C05458=1071.279,380.940,394.327,175.389,32.950,156.009
C05459=1071.272,380.693,394.366,175.385,32.942,156.008
C05460=1071.265,380.447,394.406,175.380,32.935,156.006
C05461=1071.258,380.200,394.445,175.376,32.928,156.005
C05462=1071.252,379.953,394.483,175.372,32.922,156.003
C05463=1071.245,379.706,394.522,175.368,32.915,156.002
C05464=1071.238,379.459,394.561,175.363,32.908,156.001
C05465=1071.231,379.213,394.600,175.359,32.901,155.999
C05466=1071.224,378.966,394.639,175.355,32.894,155.998
C05467=1071.217,378.719,394.678,175.350,32.887,155.996
C05468=1071.211,378.472,394.717,175.346,32.880,155.995
C05469=1071.204,378.225,394.755,175.342,32.874,155.993
C05470=1071.197,377.979,394.794,175.338,32.867,155.992
C05471=1071.190,377.732,394.833,175.333,32.860,155.990
C05472=1071.183,377.485,394.872,175.329,32.853,155.989
C05473=1071.178,377.238,394.910,175.325,32.846,155.988
C05474=1071.170,376.992,394.948,175.321,32.839,155.986
C05475=1071.163,376.745,394.987,175.316,32.832,155.985
C05476=1071.156,376.498,395.026,175.312,32.826,155.983
C05477=1071.150,376.251,395.064,175.308,32.819,155.982
C05478=1071.143,376.004,395.102,175.304,32.812,155.980
C05479=1071.136,375.757,395.141,175.300,32.806,155.979
C05480=1071.129,375.510,395.180,175.295,32.799,155.978
C05481=1071.123,375.263,395.218,175.291,32.792,155.976
C05482=1071.117,375.017,395.257,175.287,32.785,155.975
C05483=1071.110,374.770,395.296,175.283,32.779,155.973
C05484=1071.103,374.522,395.334,175.279,32.772,155.972
C05485=1071.097,374.276,395.372,175.274,32.766,155.971
C05486=1071.090,374.029,395.410,175.270,32.759,155.969
C05487=1071.083,373.782,395.449,175.266,32.753,155.968
C05488=1071.077,373.535,395.487,175.262,32.746,155.966
C05489=1071.070,373.288,395.526,175.258,32.740,155.965
C05490=1071.062,372.987,395.572,175.253,32.731,155.963
C05491=1071.054,372.685,395.619,175.248,32.723,155.962
C05492=1071.045,372.384,395.665,175.243,32.715,155.960
C05493=1071.037,372.082,395.711,175.237,32.708,155.959
C05494=1071.028,371.755,395.762,175.232,32.699,155.957
C05495=1071.019,371.427,395.812,175.227,32.691,155.955
C05496=1071.012,371.180,395.850,175.222,32.684,155.954
C05497=1071.006,370.934,395.888,175.218,32.678,155.952
C05498=1070.999,370.686,395.927,175.215,32.671,155.951
C05499=1070.992,370.439,395.964,175.211,32.665,155.950
C05500=1070.986,370.192,396.002,175.207,32.659,155.948
C05501=1070.979,369.945,396.039,175.203,32.652,155.947
C05502=1070.972,369.698,396.078,175.199,32.646,155.946
C05503=1070.966,369.452,396.115,175.195,32.640,155.944
C05504=1070.959,369.204,396.153,175.190,32.633,155.943
C05505=1070.953,368.957,396.192,175.186,32.627,155.942
C05506=1070.946,368.711,396.229,175.182,32.621,155.940
C05507=1070.939,368.463,396.267,175.178,32.614,155.939
C05508=1070.933,368.217,396.304,175.174,32.608,155.938
C05509=1070.926,367.969,396.342,175.170,32.602,155.937
C05510=1070.919,367.722,396.380,175.166,32.596,155.935
C05511=1070.913,367.475,396.417,175.162,32.589,155.934
C05512=1070.906,367.228,396.455,175.158,32.583,155.933
C05513=1070.900,366.982,396.493,175.154,32.577,155.931
C05514=1070.893,366.734,396.530,175.150,32.571,155.930
C05515=1070.887,366.487,396.567,175.146,32.564,155.929
C05516=1070.880,366.240,396.605,175.143,32.558,155.928
C05517=1070.874,365.993,396.643,175.139,32.552,155.926
C05518=1070.867,365.746,396.680,175.135,32.546,155.925
C05519=1070.861,365.499,396.718,175.131,32.539,155.924
C05520=1070.854,365.251,396.755,175.126,32.534,155.923
C05521=1070.848,365.005,396.792,175.122,32.527,155.921
C05522=1070.841,364.758,396.830,175.118,32.521,155.920
C05523=1070.835,364.510,396.867,175.114,32.515,155.919
C05524=1070.828,364.263,396.905,175.110,32.509,155.918
C05525=1070.821,364.017,396.942,175.106,32.503,155.916
C05526=1070.814,363.769,396.978,175.102,32.497,155.915
C05527=1070.808,363.522,397.016,175.098,32.490,155.914
C05528=1070.801,363.274,397.053,175.094,32.485,155.913
C05529=1070.795,363.028,397.090,175.091,32.479,155.911
C05530=1070.789,362.780,397.128,175.087,32.472,155.910
C05531=1070.782,362.533,397.165,175.083,32.467,155.909
C05532=1070.776,362.286,397.201,175.079,32.461,155.908
C05533=1070.768,362.039,397.239,175.075,32.455,155.907
C05534=1070.762,361.792,397.275,175.071,32.449,155.905
C05535=1070.756,361.545,397.313,175.067,32.443,155.904
C05536=1070.749,361.298,397.350,175.063,32.437,155.903
C05537=1070.742,361.050,397.387,175.060,32.431,155.902
C05538=1070.736,360.804,397.424,175.056,32.425,155.900
C05539=1070.729,360.557,397.460,175.052,32.419,155.899
C05540=1070.723,360.308,397.498,175.049,32.413,155.898
C05541=1070.716,360.062,397.535,175.045,32.408,155.897
C05542=1070.710,359.815,397.571,175.041,32.402,155.896
C05543=1070.703,359.567,397.608,175.037,32.396,155.895
C05544=1070.697,359.343,397.641,175.033,32.391,155.893
C05545=1070.692,359.119,397.675,175.030,32.385,155.892
C05546=1070.686,358.895,397.708,175.026,32.379,155.891
C05547=1070.680,358.671,397.741,175.023,32.374,155.890
C05548=1070.674,358.447,397.774,175.019,32.369,155.889
C05549=1070.668,358.223,397.807,175.015,32.364,155.888
C05550=1070.661,357.998,397.841,175.013,32.359,155.887
C05551=1070.656,357.774,397.875,175.009,32.354,155.886
C05552=1070.650,357.527,397.911,175.005,32.348,155.885
C05553=1070.644,357.280,397.947,175.001,32.342,155.884
C05554=1070.637,357.032,397.984,174.998,32.336,155.882
C05555=1070.630,356.786,398.020,174.994,32.331,155.881
C05556=1070.623,356.539,398.057,174.990,32.325,155.880
C05557=1070.617,356.291,398.093,174.986,32.319,155.879
C05558=1070.610,356.044,398.130,174.982,32.314,155.878
C05559=1070.604,355.797,398.166,174.979,32.308,155.877
C05560=1070.597,355.550,398.203,174.975,32.302,155.876
C05561=1070.591,355.303,398.239,174.971,32.296,155.874
C05562=1070.584,355.055,398.276,174.967,32.291,155.873
C05563=1070.578,354.807,398.312,174.964,32.285,155.872
C05564=1070.572,354.560,398.348,174.960,32.279,155.871
C05565=1070.565,354.313,398.385,174.956,32.274,155.870
C05566=1070.559,354.066,398.421,174.952,32.268,155.869
C05567=1070.553,353.819,398.457,174.949,32.262,155.868
C05568=1070.547,353.571,398.493,174.945,32.256,155.867
C05569=1070.540,353.323,398.530,174.941,32.251,155.866
C05570=1070.533,353.077,398.566,174.938,32.245,155.864
C05571=1070.527,352.829,398.602,174.934,32.240,155.863
C05572=1070.520,352.582,398.638,174.930,32.234,155.862
C05573=1070.514,352.335,398.674,174.926,32.229,155.861
C05574=1070.508,352.087,398.710,174.923,32.223,155.860
C05575=1070.502,351.840,398.747,174.919,32.217,155.859
C05576=1070.494,351.593,398.782,174.916,32.212,155.858
C05577=1070.488,351.346,398.818,174.912,32.207,155.857
C05578=1070.482,351.098,398.855,174.908,32.201,155.856
C05579=1070.475,350.851,398.890,174.904,32.195,155.854
C05580=1070.468,350.604,398.927,174.900,32.190,155.853
C05581=1070.462,350.356,398.962,174.897,32.184,155.852
C05582=1070.455,350.109,398.998,174.894,32.179,155.851
C05583=1070.449,349.862,399.034,174.890,32.174,155.850
C05584=1070.443,349.614,399.070,174.886,32.168,155.849
C05585=1070.437,349.367,399.106,174.882,32.163,155.848
C05586=1070.430,349.119,399.141,174.878,32.157,155.847
C05587=1070.424,348.872,399.177,174.875,32.152,155.846
C05588=1070.417,348.625,399.213,174.872,32.146,155.845
C05589=1070.411,348.377,399.249,174.868,32.141,155.844
C05590=1070.405,348.130,399.284,174.864,32.136,155.843
C05591=1070.398,347.883,399.320,174.861,32.130,155.842
C05592=1070.392,347.635,399.356,174.857,32.125,155.840
C05593=1070.386,347.388,399.392,174.853,32.119,155.839
C05594=1070.379,347.140,399.427,174.849,32.114,155.838
C05595=1070.373,346.893,399.463,174.847,32.109,155.837
C05596=1070.366,346.646,399.498,174.843,32.103,155.836
C05597=1070.360,346.398,399.534,174.839,32.098,155.835
C05598=1070.354,346.151,399.569,174.835,32.093,155.834
C05599=1070.348,345.904,399.604,174.832,32.087,155.833
C05600=1070.342,345.681,399.637,174.828,32.083,155.832
C05601=1070.336,345.459,399.668,174.825,32.078,155.831
C05602=1070.331,345.237,399.700,174.823,32.073,155.830
C05603=1070.325,345.014,399.732,174.819,32.068,155.829
C05604=1070.319,344.792,399.764,174.816,32.064,155.828
C05605=1070.314,344.570,399.796,174.812,32.059,155.828
C05606=1070.307,344.347,399.827,174.809,32.054,155.827
C05607=1070.302,344.125,399.859,174.806,32.049,155.826
C05608=1070.296,343.877,399.895,174.803,32.044,155.825
C05609=1070.289,343.630,399.930,174.799,32.038,155.824
C05610=1070.283,343.383,399.965,174.796,32.033,155.823
C05611=1070.277,343.136,400.000,174.792,32.028,155.822
C05612=1070.270,342.888,400.035,174.788,32.023,155.821
C05613=1070.263,342.641,400.071,174.785,32.018,155.819
C05614=1070.257,342.393,400.106,174.782,32.013,155.819
C05615=1070.251,342.145,400.141,174.778,32.007,155.818
C05616=1070.244,341.898,400.176,174.774,32.002,155.816
C05617=1070.238,341.651,400.211,174.771,31.997,155.816
C05618=1070.232,341.403,400.246,174.767,31.992,155.814
C05619=1070.225,341.155,400.281,174.763,31.986,155.813
C05620=1070.219,340.908,400.317,174.761,31.982,155.812
C05621=1070.212,340.660,400.352,174.757,31.976,155.811
C05622=1070.206,340.414,400.386,174.753,31.971,155.811
C05623=1070.200,340.166,400.421,174.750,31.966,155.809
C05624=1070.194,339.918,400.457,174.746,31.961,155.808
C05625=1070.188,339.671,400.491,174.742,31.956,155.808
C05626=1070.181,339.423,400.526,174.740,31.950,155.806
C05627=1070.175,339.176,400.561,174.736,31.946,155.806
C05628=1070.169,338.928,400.596,174.732,31.940,155.804
C05629=1070.162,338.681,400.631,174.729,31.935,155.804
C05630=1070.156,338.433,400.665,174.725,31.930,155.803
C05631=1070.150,338.185,400.701,174.722,31.925,155.802
C05632=1070.144,337.938,400.735,174.719,31.920,155.801
C05633=1070.137,337.691,400.770,174.715,31.915,155.800
C05634=1070.131,337.443,400.804,174.712,31.910,155.799
C05635=1070.125,337.196,400.839,174.708,31.905,155.798
C05636=1070.118,336.948,400.874,174.704,31.900,155.797
C05637=1070.112,336.701,400.909,174.702,31.895,155.796
C05638=1070.106,336.454,400.943,174.698,31.890,155.795
C05639=1070.099,336.206,400.977,174.695,31.885,155.794
C05640=1070.092,335.958,401.012,174.691,31.880,155.793
C05641=1070.087,335.711,401.046,174.687,31.875,155.792
C05642=1070.080,335.463,401.081,174.685,31.870,155.791
C05643=1070.074,335.215,401.117,174.681,31.865,155.790
C05644=1070.068,334.968,401.151,174.678,31.860,155.789
C05645=1070.062,334.720,401.185,174.674,31.855,155.788
C05646=1070.056,334.473,401.219,174.670,31.850,155.787
C05647=1070.049,334.225,401.254,174.667,31.845,155.786
C05648=1070.043,333.977,401.289,174.664,31.840,155.785
C05649=1070.037,333.730,401.323,174.661,31.835,155.784
C05650=1070.030,333.482,401.357,174.657,31.830,155.783
C05651=1070.024,333.235,401.391,174.654,31.825,155.782
C05652=1070.017,332.987,401.425,174.650,31.820,155.781
C05653=1070.011,332.740,401.460,174.647,31.815,155.781
C05654=1070.005,332.492,401.494,174.644,31.810,155.779
C05655=1069.999,332.245,401.528,174.640,31.805,155.779
C05656=1069.993,332.020,401.560,174.637,31.801,155.778
C05657=1069.987,331.795,401.591,174.634,31.797,155.777
C05658=1069.981,331.570,401.622,174.632,31.792,155.776
C05659=1069.977,331.345,401.653,174.628,31.788,155.775
C05660=1069.971,331.121,401.684,174.625,31.783,155.774
C05661=1069.965,330.896,401.715,174.622,31.779,155.773
C05662=1069.959,330.671,401.746,174.619,31.774,155.773
C05663=1069.953,330.446,401.777,174.617,31.770,155.772
C05664=1069.947,330.199,401.811,174.613,31.765,155.771
C05665=1069.940,329.951,401.844,174.609,31.760,155.770
C05666=1069.934,329.703,401.878,174.606,31.755,155.769
C05667=1069.928,329.455,401.912,174.602,31.751,155.768
C05668=1069.921,329.208,401.946,174.600,31.746,155.767
C05669=1069.915,328.960,401.980,174.596,31.741,155.766
C05670=1069.908,328.713,402.014,174.593,31.737,155.766
C05671=1069.902,328.465,402.047,174.589,31.732,155.765
C05672=1069.896,328.217,402.081,174.586,31.727,155.764
C05673=1069.889,327.970,402.115,174.583,31.722,155.763
C05674=1069.883,327.723,402.149,174.580,31.718,155.762
C05675=1069.876,327.474,402.182,174.576,31.713,155.761
C05676=1069.870,327.227,402.217,174.573,31.708,155.760
C05677=1069.864,326.979,402.251,174.569,31.704,155.759
C05678=1069.858,326.731,402.284,174.567,31.699,155.758
C05679=1069.852,326.484,402.318,174.563,31.694,155.758
C05680=1069.845,326.236,402.352,174.560,31.689,155.757
C05681=1069.839,325.989,402.385,174.556,31.685,155.756
C05682=1069.832,325.741,402.419,174.553,31.680,155.755
C05683=1069.826,325.493,402.452,174.550,31.675,155.754
C05684=1069.820,325.246,402.486,174.547,31.670,155.753
C05685=1069.813,324.998,402.520,174.543,31.666,155.752
C05686=1069.808,324.750,402.553,174.540,31.661,155.751
C05687=1069.801,324.503,402.587,174.537,31.656,155.750
C05688=1069.795,324.254,402.620,174.534,31.652,155.750
C05689=1069.788,324.008,402.654,174.531,31.647,155.749
C05690=1069.783,323.760,402.687,174.527,31.642,155.748
C05691=1069.776,323.512,402.721,174.524,31.638,155.747
C05692=1069.770,323.264,402.754,174.521,31.633,155.746
C05693=1069.764,323.016,402.787,174.518,31.628,155.745
C05694=1069.758,322.769,402.821,174.514,31.624,155.744
C05695=1069.751,322.521,402.854,174.511,31.619,155.743
C05696=1069.745,322.274,402.888,174.507,31.614,155.743
C05697=1069.739,322.026,402.921,174.505,31.610,155.742
C05698=1069.733,321.778,402.954,174.502,31.605,155.741
C05699=1069.726,321.530,402.988,174.498,31.600,155.740
C05700=1069.721,321.283,403.022,174.495,31.596,155.739
C05701=1069.714,321.035,403.054,174.492,31.591,155.738
C05702=1069.709,320.787,403.088,174.489,31.586,155.737
C05703=1069.702,320.540,403.121,174.486,31.582,155.736
C05704=1069.697,320.292,403.154,174.482,31.577,155.736
C05705=1069.690,320.044,403.188,174.479,31.572,155.735
C05706=1069.684,319.796,403.221,174.476,31.567,155.734
C05707=1069.677,319.549,403.254,174.473,31.563,155.733
C05708=1069.671,319.301,403.287,174.470,31.558,155.732
C05709=1069.666,319.053,403.320,174.466,31.554,155.731
C05710=1069.659,318.806,403.353,174.464,31.549,155.730
C05711=1069.654,318.558,403.387,174.460,31.545,155.730
C05712=1069.648,318.330,403.417,174.457,31.540,155.729
C05713=1069.642,318.102,403.448,174.454,31.536,155.728
C05714=1069.636,317.874,403.479,174.451,31.532,155.727
C05715=1069.631,317.647,403.508,174.449,31.528,155.726
C05716=1069.625,317.419,403.539,174.446,31.523,155.726
C05717=1069.619,317.190,403.569,174.443,31.519,155.725
C05718=1069.614,316.963,403.600,174.440,31.515,155.724
C05719=1069.609,316.735,403.630,174.438,31.511,155.723
C05720=1069.603,316.487,403.663,174.434,31.506,155.722
C05721=1069.597,316.239,403.696,174.431,31.501,155.722
C05722=1069.590,315.992,403.729,174.428,31.497,155.721
C05723=1069.585,315.744,403.762,174.425,31.492,155.720
C05724=1069.579,315.496,403.795,174.422,31.488,155.719
C05725=1069.572,315.249,403.828,174.419,31.483,155.718
C05726=1069.567,315.001,403.861,174.415,31.479,155.717
C05727=1069.560,314.753,403.894,174.412,31.474,155.716
C05728=1069.554,314.505,403.926,174.410,31.469,155.716
C05729=1069.549,314.257,403.959,174.406,31.465,155.715
C05730=1069.543,314.009,403.992,174.403,31.460,155.714
C05731=1069.536,313.762,404.024,174.400,31.456,155.713
C05732=1069.530,313.514,404.057,174.397,31.452,155.712
C05733=1069.524,313.266,404.089,174.394,31.447,155.711
C05734=1069.517,313.019,404.121,174.390,31.443,155.711
C05735=1069.511,312.771,404.154,174.387,31.438,155.710
C05736=1069.505,312.523,404.186,174.385,31.434,155.709
C05737=1069.498,312.275,404.219,174.381,31.429,155.708
C05738=1069.492,312.028,404.252,174.378,31.425,155.707
C05739=1069.486,311.779,404.284,174.375,31.421,155.707
C05740=1069.480,311.532,404.316,174.372,31.416,155.706
C05741=1069.474,311.284,404.349,174.369,31.412,155.705
C05742=1069.468,311.036,404.381,174.366,31.408,155.704
C05743=1069.461,310.789,404.413,174.362,31.403,155.703
C05744=1069.455,310.541,404.445,174.360,31.399,155.703
C05745=1069.448,310.293,404.478,174.357,31.394,155.702
C05746=1069.442,310.045,404.511,174.354,31.390,155.701
C05747=1069.436,309.797,404.543,174.350,31.385,155.700
C05748=1069.430,309.550,404.576,174.347,31.381,155.699
C05749=1069.424,309.301,404.608,174.345,31.377,155.699
C05750=1069.417,309.054,404.640,174.341,31.372,155.698
C05751=1069.411,308.806,404.672,174.338,31.368,155.697
C05752=1069.405,308.558,404.704,174.335,31.364,155.696
C05753=1069.398,308.310,404.737,174.332,31.359,155.695
C05754=1069.393,308.063,404.768,174.329,31.355,155.695
C05755=1069.387,307.815,404.801,174.326,31.351,155.694
C05756=1069.380,307.567,404.832,174.323,31.346,155.693
C05757=1069.374,307.319,404.864,174.320,31.342,155.692
C05758=1069.368,307.071,404.897,174.317,31.338,155.691
C05759=1069.362,306.823,404.929,174.314,31.333,155.691
C05760=1069.356,306.576,404.962,174.310,31.329,155.690
C05761=1069.349,306.328,404.993,174.308,31.324,155.689
C05762=1069.343,306.080,405.025,174.305,31.320,155.688
C05763=1069.337,305.832,405.057,174.302,31.315,155.687
C05764=1069.331,305.584,405.090,174.299,31.311,155.687
C05765=1069.325,305.337,405.121,174.296,31.307,155.686
C05766=1069.319,305.089,405.153,174.293,31.302,155.685
C05767=1069.313,304.841,405.185,174.290,31.298,155.684
C05768=1069.308,304.615,405.215,174.287,31.294,155.684
C05769=1069.301,304.389,405.244,174.285,31.291,155.683
C05770=1069.296,304.162,405.272,174.282,31.286,155.682
C05771=1069.291,303.936,405.302,174.279,31.282,155.681
C05772=1069.285,303.710,405.331,174.276,31.278,155.681
C05773=1069.280,303.484,405.360,174.274,31.274,155.680
C05774=1069.274,303.259,405.389,174.271,31.271,155.679
C05775=1069.269,303.032,405.418,174.268,31.266,155.678
C05776=1069.263,302.784,405.450,174.265,31.262,155.678
C05777=1069.256,302.536,405.482,174.263,31.258,155.677
C05778=1069.251,302.289,405.513,174.259,31.253,155.676
C05779=1069.245,302.041,405.545,174.256,31.249,155.675
C05780=1069.239,301.792,405.577,174.253,31.245,155.675
C05781=1069.232,301.545,405.609,174.251,31.240,155.674
C05782=1069.227,301.297,405.641,174.248,31.236,155.673
C05783=1069.221,301.049,405.673,174.244,31.231,155.672
C05784=1069.214,300.802,405.704,174.242,31.227,155.671
C05785=1069.208,300.553,405.736,174.239,31.223,155.671
C05786=1069.203,300.306,405.767,174.236,31.219,155.670
C05787=1069.196,300.058,405.799,174.233,31.214,155.669
C05788=1069.190,299.810,405.831,174.230,31.210,155.668
C05789=1069.185,299.562,405.862,174.227,31.205,155.667
C05790=1069.179,299.314,405.893,174.224,31.202,155.667
C05791=1069.173,299.066,405.925,174.221,31.197,155.666
C05792=1069.167,298.818,405.957,174.219,31.193,155.665
C05793=1069.161,298.571,405.988,174.216,31.189,155.664
C05794=1069.155,298.323,406.020,174.212,31.184,155.664
C05795=1069.150,298.075,406.052,174.209,31.180,155.663
C05796=1069.143,297.827,406.082,174.207,31.176,155.662
C05797=1069.137,297.578,406.114,174.204,31.171,155.661
C05798=1069.132,297.331,406.146,174.201,31.167,155.660
C05799=1069.125,297.083,406.177,174.199,31.163,155.660
C05800=1069.119,296.835,406.208,174.195,31.158,155.659
C05801=1069.113,296.587,406.240,174.192,31.154,155.658
C05802=1069.107,296.340,406.271,174.189,31.150,155.657
C05803=1069.102,296.091,406.302,174.187,31.146,155.657
C05804=1069.095,295.843,406.334,174.184,31.141,155.656
C05805=1069.089,295.596,406.365,174.181,31.137,155.655
C05806=1069.083,295.347,406.396,174.177,31.133,155.654
C05807=1069.077,295.100,406.427,174.175,31.129,155.654
C05808=1069.070,294.851,406.458,174.172,31.124,155.653
C05809=1069.065,294.604,406.489,174.169,31.121,155.652
C05810=1069.059,294.355,406.520,174.166,31.116,155.651
C05811=1069.053,294.108,406.551,174.164,31.112,155.651
C05812=1069.047,293.860,406.583,174.161,31.108,155.650
C05813=1069.041,293.612,406.614,174.157,31.104,155.649
C05814=1069.034,293.364,406.645,174.155,31.099,155.648
C05815=1069.028,293.116,406.675,174.152,31.095,155.648
C05816=1069.022,292.867,406.707,174.149,31.091,155.647
C05817=1069.016,292.620,406.738,174.146,31.087,155.646
C05818=1069.010,292.372,406.769,174.144,31.083,155.645
C05819=1069.004,292.124,406.800,174.141,31.079,155.645
C05820=1068.998,291.876,406.831,174.138,31.074,155.644
C05821=1068.992,291.628,406.862,174.136,31.070,155.643
C05822=1068.986,291.380,406.893,174.132,31.066,155.642
C05823=1068.980,291.132,406.923,174.129,31.062,155.642
C05824=1068.975,290.913,406.951,174.127,31.058,155.641
C05825=1068.969,290.694,406.978,174.125,31.054,155.640
C05826=1068.963,290.476,407.005,174.122,31.051,155.640
C05827=1068.958,290.258,407.032,174.119,31.047,155.639
C05828=1068.954,290.038,407.059,174.117,31.044,155.638
C05829=1068.948,289.820,407.086,174.115,31.040,155.638
C05830=1068.942,289.601,407.113,174.112,31.036,155.637
C05831=1068.937,289.382,407.141,174.109,31.032,155.636
C05832=1068.932,289.134,407.172,174.106,31.028,155.636
C05833=1068.926,288.886,407.202,174.104,31.024,155.635
C05834=1068.919,288.639,407.233,174.101,31.020,155.634
C05835=1068.913,288.391,407.264,174.098,31.016,155.634
C05836=1068.907,288.142,407.294,174.095,31.012,155.633
C05837=1068.901,287.894,407.325,174.093,31.007,155.632
C05838=1068.895,287.646,407.355,174.090,31.004,155.631
C05839=1068.889,287.398,407.386,174.087,30.999,155.631
C05840=1068.883,287.150,407.416,174.085,30.995,155.630
C05841=1068.876,286.902,407.447,174.082,30.991,155.629
C05842=1068.871,286.654,407.477,174.079,30.987,155.628
C05843=1068.865,286.406,407.508,174.076,30.983,155.628
C05844=1068.858,286.158,407.539,174.073,30.979,155.627
C05845=1068.852,285.910,407.569,174.070,30.975,155.626
C05846=1068.846,285.662,407.600,174.067,30.971,155.626
C05847=1068.840,285.414,407.630,174.065,30.966,155.625
C05848=1068.834,285.166,407.661,174.062,30.962,155.624
C05849=1068.828,284.918,407.690,174.059,30.958,155.623
C05850=1068.822,284.669,407.721,174.057,30.954,155.622
C05851=1068.816,284.422,407.751,174.054,30.950,155.622
C05852=1068.810,284.174,407.781,174.051,30.946,155.621
C05853=1068.804,283.925,407.812,174.048,30.942,155.620
C05854=1068.798,283.677,407.842,174.046,30.938,155.620
C05855=1068.792,283.430,407.873,174.043,30.934,155.619
C05856=1068.786,283.182,407.903,174.040,30.929,155.618
C05857=1068.780,282.933,407.934,174.038,30.926,155.617
C05858=1068.774,282.685,407.964,174.035,30.921,155.617
C05859=1068.768,282.437,407.994,174.032,30.917,155.616
C05860=1068.763,282.189,408.024,174.029,30.913,155.615
C05861=1068.755,281.941,408.054,174.027,30.909,155.614
C05862=1068.750,281.693,408.085,174.024,30.905,155.614
C05863=1068.744,281.445,408.114,174.021,30.900,155.613
C05864=1068.738,281.197,408.145,174.019,30.897,155.612
C05865=1068.732,280.949,408.175,174.016,30.892,155.612
C05866=1068.726,280.701,408.206,174.013,30.888,155.611
C05867=1068.720,280.452,408.235,174.011,30.884,155.610
C05868=1068.714,280.205,408.265,174.008,30.880,155.609
C05869=1068.708,279.957,408.295,174.005,30.876,155.609
C05870=1068.703,279.708,408.325,174.002,30.872,155.608
C05871=1068.696,279.460,408.356,174.000,30.868,155.607
C05872=1068.690,279.212,408.385,173.997,30.864,155.607
C05873=1068.684,278.964,408.415,173.994,30.860,155.606
C05874=1068.678,278.716,408.445,173.992,30.856,155.605
C05875=1068.672,278.468,408.474,173.989,30.852,155.604
C05876=1068.666,278.219,408.505,173.986,30.848,155.604
C05877=1068.660,277.971,408.535,173.983,30.844,155.603
C05878=1068.654,277.723,408.565,173.981,30.839,155.602
C05879=1068.648,277.476,408.595,173.978,30.835,155.602
C05880=1068.643,277.261,408.620,173.975,30.832,155.601
C05881=1068.638,277.048,408.646,173.974,30.829,155.600
C05882=1068.632,276.834,408.672,173.971,30.825,155.600
C05883=1068.628,276.621,408.697,173.969,30.822,155.599
C05884=1068.622,276.407,408.723,173.966,30.818,155.598
C05885=1068.617,276.194,408.748,173.965,30.815,155.598
C05886=1068.611,275.980,408.774,173.962,30.811,155.597
C05887=1068.607,275.767,408.800,173.960,30.808,155.597
C05888=1068.601,275.518,408.829,173.957,30.803,155.596
C05889=1068.595,275.271,408.859,173.955,30.800,155.595
C05890=1068.589,275.022,408.889,173.952,30.795,155.594
C05891=1068.583,274.774,408.918,173.949,30.791,155.594
C05892=1068.576,274.526,408.949,173.947,30.788,155.593
C05893=1068.570,274.278,408.978,173.944,30.783,155.592
C05894=1068.565,274.029,409.007,173.941,30.779,155.592
C05895=1068.558,273.782,409.037,173.939,30.775,155.591
C05896=1068.553,273.533,409.067,173.936,30.771,155.590
C05897=1068.547,273.285,409.096,173.933,30.767,155.590
C05898=1068.540,273.037,409.126,173.931,30.763,155.589
C05899=1068.535,272.789,409.156,173.928,30.759,155.588
C05900=1068.529,272.541,409.185,173.925,30.755,155.587
C05901=1068.522,272.293,409.214,173.923,30.751,155.587
C05902=1068.517,272.044,409.243,173.920,30.747,155.586
C05903=1068.510,271.797,409.273,173.918,30.743,155.585
C05904=1068.505,271.548,409.303,173.915,30.739,155.585
C05905=1068.499,271.300,409.332,173.913,30.735,155.584
C05906=1068.493,271.052,409.361,173.910,30.731,155.583
C05907=1068.487,270.804,409.391,173.907,30.727,155.583
C05908=1068.481,270.555,409.420,173.905,30.723,155.582
C05909=1068.475,270.307,409.449,173.902,30.719,155.581
C05910=1068.469,270.059,409.478,173.899,30.715,155.580
C05911=1068.462,269.811,409.508,173.897,30.710,155.580
C05912=1068.457,269.563,409.538,173.894,30.707,155.579
C05913=1068.451,269.315,409.567,173.891,30.703,155.578
C05914=1068.445,269.066,409.596,173.889,30.698,155.578
C05915=1068.439,268.818,409.625,173.887,30.695,155.577
C05916=1068.433,268.570,409.654,173.884,30.691,155.576
C05917=1068.426,268.322,409.683,173.882,30.686,155.575
C05918=1068.421,268.073,409.713,173.879,30.683,155.575
C05919=1068.415,267.825,409.742,173.876,30.679,155.574
C05920=1068.409,267.577,409.770,173.873,30.675,155.573
C05921=1068.402,267.328,409.799,173.871,30.670,155.573
C05922=1068.397,267.080,409.829,173.868,30.667,155.572
C05923=1068.391,266.832,409.858,173.865,30.663,155.571
C05924=1068.384,266.584,409.887,173.864,30.659,155.571
C05925=1068.378,266.336,409.916,173.861,30.655,155.570
C05926=1068.373,266.087,409.946,173.858,30.651,155.569
C05927=1068.366,265.839,409.975,173.856,30.646,155.569
C05928=1068.360,265.590,410.003,173.853,30.643,155.568
C05929=1068.355,265.343,410.032,173.850,30.639,155.567
C05930=1068.349,265.094,410.062,173.848,30.634,155.566
C05931=1068.343,264.846,410.091,173.845,30.631,155.566
C05932=1068.337,264.598,410.120,173.843,30.627,155.565
C05933=1068.331,264.349,410.148,173.841,30.622,155.564
C05934=1068.325,264.101,410.177,173.838,30.619,155.564
C05935=1068.319,263.853,410.207,173.835,30.615,155.563
C05936=1068.314,263.642,410.230,173.834,30.611,155.562
C05937=1068.309,263.429,410.255,173.831,30.608,155.562
C05938=1068.304,263.218,410.280,173.829,30.605,155.561
C05939=1068.298,263.006,410.304,173.826,30.601,155.561
C05940=1068.293,262.794,410.329,173.825,30.598,155.560
C05941=1068.287,262.582,410.353,173.822,30.594,155.559
C05942=1068.283,262.370,410.378,173.820,30.591,155.559
C05943=1068.277,262.159,410.402,173.819,30.588,155.558
C05944=1068.271,261.910,410.431,173.816,30.584,155.558
C05945=1068.264,261.662,410.460,173.813,30.580,155.557
C05946=1068.259,261.414,410.488,173.811,30.576,155.556
C05947=1068.253,261.166,410.517,173.808,30.572,155.556
C05948=1068.247,260.917,410.546,173.805,30.568,155.555
C05949=1068.241,260.669,410.574,173.803,30.564,155.554
C05950=1068.234,260.421,410.603,173.801,30.560,155.554
C05951=1068.228,260.172,410.631,173.798,30.556,155.553
C05952=1068.221,259.924,410.660,173.795,30.552,155.552
C05953=1068.216,259.676,410.688,173.793,30.548,155.551
C05954=1068.210,259.427,410.716,173.790,30.544,155.551
C05955=1068.204,259.179,410.745,173.788,30.540,155.550
C05956=1068.198,258.930,410.774,173.786,30.537,155.549
C05957=1068.192,258.682,410.803,173.783,30.533,155.549
C05958=1068.186,258.434,410.831,173.780,30.528,155.548
C05959=1068.179,258.186,410.859,173.778,30.524,155.547
C05960=1068.173,257.938,410.887,173.775,30.521,155.547
C05961=1068.167,257.689,410.916,173.773,30.517,155.546
C05962=1068.161,257.441,410.945,173.771,30.513,155.545
C05963=1068.156,257.193,410.973,173.768,30.509,155.545
C05964=1068.150,256.944,411.001,173.765,30.505,155.544
C05965=1068.144,256.696,411.030,173.763,30.501,155.543
C05966=1068.137,256.447,411.058,173.761,30.497,155.543
C05967=1068.132,256.199,411.086,173.759,30.493,155.542
C05968=1068.125,255.951,411.115,173.756,30.489,155.541
C05969=1068.119,255.702,411.143,173.753,30.485,155.541
C05970=1068.114,255.454,411.171,173.751,30.481,155.540
C05971=1068.107,255.206,411.199,173.749,30.477,155.539
C05972=1068.101,254.958,411.228,173.746,30.473,155.538
C05973=1068.095,254.709,411.256,173.744,30.469,155.538
C05974=1068.090,254.461,411.284,173.741,30.465,155.537
C05975=1068.084,254.212,411.312,173.739,30.461,155.536
C05976=1068.077,253.964,411.340,173.737,30.457,155.536
C05977=1068.072,253.716,411.369,173.734,30.453,155.535
C05978=1068.066,253.468,411.397,173.731,30.449,155.534
C05979=1068.060,253.219,411.425,173.730,30.445,155.534
C05980=1068.054,252.971,411.453,173.727,30.441,155.533
C05981=1068.048,252.722,411.481,173.724,30.437,155.532
C05982=1068.042,252.474,411.509,173.722,30.433,155.532
C05983=1068.036,252.226,411.537,173.720,30.429,155.531
C05984=1068.031,251.977,411.566,173.717,30.425,155.530
C05985=1068.024,251.729,411.593,173.715,30.421,155.529
C05986=1068.019,251.480,411.621,173.712,30.417,155.529
C05987=1068.013,251.232,411.649,173.710,30.413,155.528
C05988=1068.007,250.983,411.678,173.708,30.410,155.527
C05989=1068.001,250.735,411.705,173.705,30.405,155.527
C05990=1067.995,250.487,411.733,173.702,30.401,155.526
C05991=1067.989,250.238,411.762,173.701,30.397,155.525
C05992=1067.984,250.026,411.786,173.698,30.394,155.525
C05993=1067.978,249.813,411.810,173.696,30.390,155.524
C05994=1067.974,249.600,411.834,173.695,30.387,155.524
C05995=1067.969,249.387,411.858,173.692,30.383,155.523
C05996=1067.964,249.174,411.882,173.690,30.380,155.522
C05997=1067.959,248.961,411.906,173.689,30.377,155.522
C05998=1067.954,248.748,411.929,173.686,30.373,155.521
C05999=1067.949,248.535,411.954,173.684,30.370,155.521
C06000=1067.943,248.287,411.982,173.682,30.366,155.520
C06001=1067.938,248.037,412.009,173.679,30.361,155.519
C06002=1067.932,247.790,412.037,173.677,30.358,155.518
C06003=1067.926,247.541,412.065,173.675,30.354,155.518
C06004=1067.920,247.293,412.093,173.672,30.349,155.517
C06005=1067.914,247.045,412.121,173.670,30.345,155.516
C06006=1067.908,246.796,412.149,173.668,30.342,155.516
C06007=1067.903,246.547,412.176,173.665,30.337,155.515
C06008=1067.897,246.299,412.204,173.663,30.333,155.514
C06009=1067.891,246.051,412.232,173.661,30.330,155.514
C06010=1067.885,245.803,412.259,173.658,30.326,155.513
C06011=1067.879,245.553,412.287,173.656,30.321,155.512
C06012=1067.873,245.306,412.314,173.654,30.318,155.512
C06013=1067.867,245.057,412.343,173.651,30.314,155.511
C06014=1067.861,244.809,412.369,173.649,30.309,155.510
C06015=1067.854,244.560,412.397,173.647,30.305,155.509
C06016=1067.849,244.312,412.425,173.644,30.302,155.509
C06017=1067.843,244.063,412.452,173.642,30.298,155.508
C06018=1067.837,243.815,412.480,173.640,30.293,155.507
C06019=1067.831,243.567,412.508,173.637,30.290,155.507
C06020=1067.826,243.318,412.535,173.635,30.286,155.506
C06021=1067.820,243.070,412.562,173.633,30.281,155.505
C06022=1067.814,242.821,412.590,173.631,30.277,155.505
C06023=1067.808,242.573,412.617,173.628,30.274,155.504
C06024=1067.801,242.325,412.645,173.626,30.270,155.503
C06025=1067.796,242.076,412.672,173.624,30.265,155.503
C06026=1067.790,241.828,412.700,173.621,30.261,155.502
C06027=1067.784,241.579,412.727,173.619,30.258,155.501
C06028=1067.778,241.330,412.755,173.617,30.254,155.501
C06029=1067.772,241.082,412.781,173.614,30.249,155.500
C06030=1067.766,240.834,412.808,173.613,30.246,155.499
C06031=1067.760,240.585,412.836,173.610,30.242,155.499
C06032=1067.755,240.337,412.863,173.607,30.238,155.498
C06033=1067.748,240.088,412.891,173.606,30.234,155.497
C06034=1067.742,239.840,412.917,173.603,30.230,155.496
C06035=1067.735,239.591,412.945,173.600,30.226,155.496
C06036=1067.730,239.343,412.972,173.599,30.222,155.495
C06037=1067.725,239.094,412.999,173.596,30.218,155.494
C06038=1067.718,238.846,413.027,173.594,30.214,155.494
C06039=1067.712,238.597,413.053,173.592,30.210,155.493
C06040=1067.706,238.349,413.080,173.589,30.206,155.492
C06041=1067.700,238.101,413.108,173.587,30.202,155.492
C06042=1067.695,237.852,413.135,173.585,30.198,155.491
C06043=1067.688,237.603,413.162,173.582,30.194,155.490
C06044=1067.682,237.355,413.189,173.580,30.190,155.490
C06045=1067.676,237.107,413.216,173.578,30.186,155.489
C06046=1067.670,236.858,413.243,173.576,30.182,155.488
C06047=1067.664,236.609,413.270,173.574,30.178,155.488
C06048=1067.660,236.394,413.294,173.571,30.175,155.487
C06049=1067.654,236.177,413.317,173.570,30.171,155.486
C06050=1067.649,235.961,413.341,173.568,30.168,155.486
C06051=1067.644,235.745,413.364,173.565,30.164,155.485
C06052=1067.638,235.529,413.387,173.564,30.161,155.485
C06053=1067.634,235.313,413.411,173.562,30.157,155.484
C06054=1067.628,235.097,413.435,173.560,30.154,155.483
C06055=1067.624,234.880,413.458,173.558,30.150,155.483
C06056=1067.617,234.631,413.485,173.556,30.146,155.482
C06057=1067.612,234.383,413.512,173.553,30.142,155.481
C06058=1067.606,234.135,413.539,173.551,30.139,155.481
C06059=1067.600,233.887,413.566,173.549,30.134,155.480
C06060=1067.593,233.638,413.593,173.546,30.130,155.479
C06061=1067.588,233.389,413.619,173.545,30.127,155.479
C06062=1067.582,233.141,413.646,173.542,30.122,155.478
C06063=1067.575,232.892,413.673,173.540,30.118,155.477
C06064=1067.570,232.643,413.700,173.538,30.114,155.477
C06065=1067.564,232.395,413.726,173.535,30.110,155.476
C06066=1067.558,232.147,413.753,173.534,30.106,155.475
C06067=1067.552,231.898,413.780,173.531,30.102,155.475
C06068=1067.546,231.649,413.807,173.529,30.098,155.474
C06069=1067.540,231.401,413.833,173.527,30.094,155.473
C06070=1067.534,231.153,413.860,173.524,30.090,155.472
C06071=1067.529,230.904,413.886,173.523,30.086,155.472
C06072=1067.522,230.655,413.914,173.520,30.082,155.471
C06073=1067.517,230.407,413.940,173.519,30.078,155.470
C06074=1067.511,230.158,413.967,173.516,30.074,155.470
C06075=1067.505,229.910,413.993,173.513,30.070,155.469
C06076=1067.499,229.662,414.020,173.512,30.066,155.468
C06077=1067.493,229.412,414.046,173.509,30.062,155.468
C06078=1067.487,229.164,414.072,173.507,30.058,155.467
C06079=1067.481,228.916,414.099,173.505,30.055,155.466
C06080=1067.475,228.667,414.126,173.503,30.050,155.466
C06081=1067.469,228.418,414.153,173.501,30.046,155.465
C06082=1067.463,228.170,414.179,173.498,30.042,155.464
C06083=1067.457,227.921,414.205,173.496,30.039,155.464
C06084=1067.451,227.673,414.231,173.494,30.034,155.463
C06085=1067.445,227.425,414.258,173.492,30.030,155.462
C06086=1067.439,227.176,414.285,173.490,30.027,155.462
C06087=1067.433,226.927,414.310,173.488,30.022,155.461
C06088=1067.427,226.678,414.337,173.485,30.018,155.460
C06089=1067.421,226.430,414.364,173.484,30.015,155.459
C06090=1067.415,226.182,414.390,173.481,30.011,155.459
C06091=1067.409,225.933,414.416,173.479,30.006,155.458
C06092=1067.403,225.685,414.442,173.477,30.002,155.457
C06093=1067.398,225.436,414.469,173.474,29.998,155.457
C06094=1067.391,225.187,414.495,173.473,29.994,155.456
C06095=1067.385,224.939,414.521,173.470,29.990,155.455
C06096=1067.379,224.690,414.548,173.469,29.986,155.455
C06097=1067.374,224.441,414.574,173.466,29.982,155.454
C06098=1067.368,224.193,414.601,173.464,29.978,155.453
C06099=1067.361,223.945,414.627,173.462,29.974,155.453
C06100=1067.356,223.696,414.653,173.460,29.970,155.452
C06101=1067.350,223.447,414.679,173.458,29.966,155.451
C06102=1067.344,223.199,414.705,173.456,29.962,155.450
C06103=1067.338,222.950,414.731,173.454,29.958,155.450
C06104=1067.333,222.730,414.755,173.452,29.955,155.449
C06105=1067.328,222.510,414.778,173.450,29.951,155.449
C06106=1067.322,222.290,414.800,173.448,29.948,155.448
C06107=1067.317,222.069,414.824,173.446,29.944,155.447
C06108=1067.312,221.849,414.847,173.444,29.940,155.447
C06109=1067.307,221.629,414.870,173.443,29.937,155.446
C06110=1067.301,221.409,414.893,173.440,29.933,155.445
C06111=1067.297,221.189,414.917,173.438,29.929,155.445
C06112=1067.290,220.940,414.942,173.437,29.925,155.444
C06113=1067.285,220.691,414.968,173.434,29.921,155.443
C06114=1067.278,220.443,414.994,173.433,29.918,155.443
C06115=1067.273,220.194,415.020,173.430,29.913,155.442
C06116=1067.266,219.946,415.046,173.428,29.909,155.441
C06117=1067.260,219.697,415.071,173.426,29.906,155.441
C06118=1067.255,219.448,415.097,173.424,29.901,155.440
C06119=1067.248,219.200,415.123,173.422,29.897,155.439
C06120=1067.243,218.951,415.149,173.420,29.894,155.439
C06121=1067.236,218.703,415.175,173.418,29.889,155.438
C06122=1067.231,218.454,415.201,173.416,29.885,155.437
C06123=1067.225,218.205,415.227,173.413,29.881,155.437
C06124=1067.219,217.956,415.253,173.412,29.877,155.436
C06125=1067.213,217.708,415.279,173.409,29.873,155.435
C06126=1067.207,217.459,415.305,173.408,29.869,155.435
C06127=1067.201,217.211,415.330,173.405,29.865,155.434
C06128=1067.194,216.963,415.356,173.404,29.861,155.433
C06129=1067.189,216.714,415.382,173.401,29.857,155.432
C06130=1067.183,216.465,415.407,173.399,29.853,155.432
C06131=1067.177,216.216,415.433,173.397,29.849,155.431
C06132=1067.171,215.968,415.459,173.395,29.845,155.430
C06133=1067.165,215.719,415.485,173.393,29.841,155.430
C06134=1067.159,215.470,415.511,173.391,29.837,155.429
C06135=1067.153,215.222,415.536,173.390,29.833,155.428
C06136=1067.147,214.973,415.562,173.387,29.829,155.428
C06137=1067.141,214.724,415.587,173.385,29.825,155.427
C06138=1067.136,214.476,415.614,173.383,29.820,155.426
C06139=1067.130,214.228,415.639,173.381,29.817,155.425
C06140=1067.124,213.979,415.664,173.379,29.812,155.425
C06141=1067.118,213.730,415.690,173.377,29.808,155.424
C06142=1067.112,213.481,415.715,173.374,29.804,155.423
C06143=1067.106,213.233,415.741,173.373,29.800,155.423
C06144=1067.100,212.984,415.767,173.370,29.796,155.422
C06145=1067.094,212.735,415.792,173.369,29.792,155.421
C06146=1067.089,212.487,415.817,173.367,29.788,155.421
C06147=1067.083,212.238,415.843,173.365,29.784,155.420
C06148=1067.077,211.989,415.868,173.363,29.780,155.419
C06149=1067.071,211.741,415.894,173.361,29.776,155.418
C06150=1067.064,211.492,415.919,173.359,29.771,155.418
C06151=1067.059,211.243,415.945,173.356,29.767,155.417
C06152=1067.053,210.995,415.970,173.355,29.764,155.416
C06153=1067.047,210.747,415.995,173.353,29.759,155.416
C06154=1067.041,210.498,416.020,173.351,29.755,155.415
C06155=1067.035,210.249,416.046,173.349,29.751,155.414
C06156=1067.029,210.000,416.072,173.347,29.747,155.414
C06157=1067.023,209.752,416.097,173.345,29.743,155.413
C06158=1067.017,209.503,416.122,173.343,29.739,155.412
C06159=1067.011,209.255,416.147,173.341,29.735,155.411
C06160=1067.005,209.037,416.170,173.339,29.731,155.411
C06161=1067.001,208.819,416.191,173.338,29.728,155.410
C06162=1066.995,208.601,416.213,173.336,29.724,155.410
C06163=1066.990,208.383,416.237,173.334,29.720,155.409
C06164=1066.985,208.165,416.258,173.332,29.717,155.408
C06165=1066.980,207.947,416.280,173.330,29.713,155.408
C06166=1066.975,207.729,416.303,173.329,29.710,155.407
C06167=1066.970,207.511,416.324,173.327,29.706,155.407
C06168=1066.945,206.466,416.427,173.176,29.631,155.402
C06169=1066.939,206.217,416.452,173.174,29.627,155.402
C06170=1066.934,205.969,416.476,173.171,29.624,155.401
C06171=1066.927,205.720,416.500,173.169,29.621,155.401
C06172=1066.922,205.471,416.525,173.167,29.618,155.400
C06173=1066.917,205.222,416.549,173.165,29.614,155.400
C06174=1066.911,204.973,416.573,173.162,29.611,155.399
C06175=1066.905,204.725,416.598,173.160,29.608,155.399
C06176=1066.899,204.476,416.622,173.158,29.605,155.398
C06177=1066.893,204.228,416.647,173.155,29.602,155.398
C06178=1066.887,203.978,416.671,173.154,29.599,155.397
C06179=1066.882,203.730,416.696,173.151,29.595,155.397
C06180=1066.877,203.481,416.720,173.150,29.592,155.396
C06181=1066.870,203.232,416.744,173.147,29.589,155.396
C06182=1066.865,202.984,416.768,173.144,29.586,155.395
C06183=1066.859,202.735,416.792,173.143,29.583,155.395
C06184=1066.854,202.486,416.817,173.140,29.580,155.394
C06185=1066.847,202.237,416.841,173.138,29.576,155.394
C06186=1066.842,201.988,416.865,173.136,29.573,155.393
C06187=1066.836,201.740,416.889,173.134,29.570,155.393
C06188=1066.830,201.491,416.913,173.131,29.567,155.392
C06189=1066.824,201.242,416.938,173.130,29.564,155.392
C06190=1066.818,200.994,416.961,173.127,29.561,155.391
C06191=1066.813,200.744,416.985,173.125,29.558,155.391
C06192=1066.807,200.496,417.009,173.123,29.555,155.390
C06193=1066.801,200.247,417.033,173.120,29.552,155.390
C06194=1066.795,199.998,417.057,173.119,29.549,155.390
C06195=1066.789,199.749,417.082,173.116,29.546,155.389
C06196=1066.783,199.501,417.105,173.114,29.542,155.389
C06197=1066.777,199.252,417.129,173.112,29.540,155.388
C06198=1066.772,199.003,417.153,173.110,29.536,155.388
C06199=1066.765,198.754,417.177,173.107,29.533,155.387
C06200=1066.760,198.505,417.201,173.106,29.530,155.387
C06201=1066.754,198.257,417.225,173.103,29.527,155.386
C06202=1066.748,198.008,417.249,173.102,29.524,155.386
C06203=1066.742,197.759,417.272,173.099,29.521,155.385
C06204=1066.737,197.510,417.297,173.097,29.518,155.385
C06205=1066.731,197.262,417.320,173.095,29.515,155.385
C06206=1066.725,197.013,417.345,173.092,29.512,155.384
C06207=1066.719,196.764,417.368,173.090,29.509,155.384
C06208=1066.714,196.515,417.392,173.088,29.506,155.383
C06209=1066.707,196.266,417.416,173.086,29.503,155.383
C06210=1066.702,196.018,417.440,173.083,29.499,155.382
C06211=1066.696,195.769,417.463,173.082,29.497,155.382
C06212=1066.690,195.521,417.487,173.079,29.493,155.381
C06213=1066.684,195.271,417.512,173.077,29.491,155.381
C06214=1066.679,195.022,417.534,173.075,29.487,155.380
C06215=1066.673,194.774,417.559,173.073,29.485,155.380
C06216=1066.667,194.526,417.582,173.071,29.481,155.379
C06217=1066.662,194.276,417.606,173.069,29.478,155.379
C06218=1066.656,194.027,417.630,173.067,29.475,155.378
C06219=1066.650,193.778,417.653,173.065,29.472,155.378
C06220=1066.645,193.530,417.677,173.063,29.469,155.377
C06221=1066.638,193.281,417.701,173.060,29.466,155.377
C06222=1066.633,193.032,417.725,173.059,29.463,155.377
C06223=1066.627,192.783,417.748,173.056,29.460,155.376
C06224=1066.621,192.534,417.771,173.055,29.457,155.376
C06225=1066.616,192.286,417.796,173.052,29.454,155.375
C06226=1066.610,192.037,417.819,173.050,29.451,155.375
C06227=1066.604,191.788,417.843,173.048,29.448,155.374
C06228=1066.599,191.539,417.866,173.046,29.445,155.374
C06229=1066.592,191.256,417.893,173.043,29.441,155.373
C06230=1066.586,190.974,417.920,173.041,29.438,155.373
C06231=1066.579,190.692,417.947,173.038,29.434,155.372
C06232=1066.572,190.409,417.973,173.037,29.431,155.372
C06233=1066.567,190.160,417.997,173.034,29.428,155.371
C06234=1066.562,189.911,418.020,173.032,29.425,155.371
C06235=1066.556,189.663,418.044,173.030,29.421,155.370
C06236=1066.550,189.413,418.067,173.028,29.419,155.370
C06237=1066.544,189.165,418.091,173.026,29.415,155.369
C06238=1066.539,188.915,418.115,173.024,29.413,155.369
C06239=1066.533,188.667,418.138,173.022,29.409,155.368
C06240=1066.527,188.418,418.161,173.020,29.406,155.368
C06241=1066.522,188.169,418.185,173.018,29.403,155.368
C06242=1066.516,187.921,418.208,173.015,29.400,155.367
C06243=1066.510,187.672,418.231,173.014,29.397,155.367
C06244=1066.505,187.423,418.255,173.011,29.394,155.366
C06245=1066.499,187.174,418.279,173.009,29.391,155.366
C06246=1066.494,186.926,418.301,173.008,29.388,155.365
C06247=1066.489,186.676,418.325,173.005,29.385,155.365
C06248=1066.483,186.427,418.348,173.004,29.382,155.364
C06249=1066.477,186.179,418.372,173.001,29.379,155.364
C06250=1066.472,185.930,418.395,172.999,29.376,155.363
C06251=1066.466,185.681,418.418,172.998,29.373,155.363
C06252=1066.460,185.432,418.441,172.995,29.370,155.362
C06253=1066.454,185.183,418.466,172.993,29.367,155.362
C06254=1066.449,184.934,418.489,172.991,29.364,155.362
C06255=1066.443,184.685,418.512,172.989,29.360,155.361
C06256=1066.437,184.436,418.535,172.988,29.358,155.361
C06257=1066.432,184.187,418.557,172.985,29.355,155.360
C06258=1066.426,183.939,418.581,172.983,29.352,155.360
C06259=1066.420,183.690,418.604,172.981,29.349,155.359
C06260=1066.414,183.441,418.627,172.979,29.346,155.359
C06261=1066.408,183.192,418.650,172.977,29.343,155.358
C06262=1066.402,182.944,418.672,172.975,29.340,155.358
C06263=1066.396,182.694,418.696,172.973,29.338,155.358
C06264=1066.390,182.445,418.719,172.970,29.334,155.357
C06265=1066.384,182.196,418.742,172.969,29.332,155.357
C06266=1066.378,181.947,418.764,172.967,29.329,155.356
C06267=1066.373,181.699,418.787,172.964,29.326,155.356
C06268=1066.367,181.450,418.810,172.963,29.323,155.355
C06269=1066.360,181.201,418.833,172.960,29.320,155.355
C06270=1066.355,180.952,418.856,172.959,29.317,155.355
C06271=1066.349,180.703,418.879,172.957,29.314,155.354
C06272=1066.343,180.454,418.902,172.954,29.311,155.354
C06273=1066.337,180.205,418.925,172.953,29.308,155.353
C06274=1066.332,179.957,418.947,172.950,29.305,155.353
C06275=1066.325,179.708,418.970,172.948,29.303,155.352
C06276=1066.320,179.459,418.993,172.947,29.300,155.352
C06277=1066.314,179.210,419.016,172.944,29.296,155.352
C06278=1066.308,178.961,419.039,172.942,29.294,155.351
C06279=1066.302,178.712,419.062,172.941,29.291,155.351
C06280=1066.297,178.464,419.085,172.938,29.288,155.350
C06281=1066.290,178.215,419.107,172.937,29.286,155.350
C06282=1066.284,177.966,419.130,172.935,29.282,155.349
C06283=1066.279,177.717,419.153,172.932,29.279,155.349
C06284=1066.273,177.468,419.176,172.931,29.277,155.349
C06285=1066.267,177.219,419.199,172.928,29.274,155.348
C06286=1066.261,176.970,419.220,172.926,29.270,155.348
C06287=1066.255,176.721,419.243,172.925,29.268,155.347
C06288=1066.250,176.472,419.266,172.922,29.265,155.347
C06289=1066.244,176.223,419.289,172.920,29.262,155.346
C06290=1066.238,175.975,419.312,172.919,29.259,155.346
C06291=1066.232,175.726,419.334,172.916,29.256,155.346
C06292=1066.226,175.476,419.357,172.915,29.253,155.345
C06293=1066.220,175.193,419.383,172.912,29.250,155.345
C06294=1066.213,174.910,419.409,172.910,29.247,155.344
C06295=1066.206,174.628,419.434,172.908,29.244,155.344
C06296=1066.200,174.345,419.460,172.906,29.240,155.343
C06297=1066.194,174.095,419.482,172.904,29.237,155.343
C06298=1066.189,173.847,419.505,172.902,29.234,155.342
C06299=1066.183,173.598,419.528,172.900,29.232,155.342
C06300=1066.176,173.349,419.550,172.898,29.229,155.341
C06301=1066.171,173.100,419.573,172.896,29.226,155.341
C06302=1066.166,172.851,419.595,172.894,29.223,155.341
C06303=1066.160,172.603,419.618,172.892,29.220,155.340
C06304=1066.154,172.353,419.640,172.890,29.217,155.340
C06305=1066.148,172.104,419.663,172.888,29.214,155.339
C06306=1066.142,171.856,419.686,172.886,29.211,155.339
C06307=1066.136,171.606,419.707,172.884,29.208,155.338
C06308=1066.131,171.358,419.730,172.883,29.205,155.338
C06309=1066.125,171.109,419.753,172.880,29.203,155.338
C06310=1066.120,170.860,419.775,172.878,29.199,155.337
C06311=1066.114,170.611,419.797,172.877,29.197,155.337
C06312=1066.108,170.362,419.820,172.875,29.194,155.336
C06313=1066.102,170.113,419.842,172.872,29.191,155.336
C06314=1066.097,169.865,419.864,172.871,29.188,155.335
C06315=1066.091,169.615,419.887,172.869,29.185,155.335
C06316=1066.085,169.366,419.910,172.867,29.182,155.335
C06317=1066.080,169.117,419.932,172.865,29.179,155.334
C06318=1066.074,168.869,419.954,172.863,29.176,155.334
C06319=1066.069,168.619,419.976,172.862,29.173,155.333
C06320=1066.063,168.371,419.999,172.859,29.170,155.333
C06321=1066.057,168.121,420.021,172.857,29.168,155.332
C06322=1066.051,167.872,420.044,172.856,29.165,155.332
C06323=1066.046,167.624,420.065,172.854,29.162,155.331
C06324=1066.040,167.375,420.088,172.852,29.159,155.331
C06325=1066.034,167.126,420.110,172.850,29.156,155.331
C06326=1066.029,166.877,420.133,172.848,29.153,155.330
C06327=1066.023,166.628,420.154,172.846,29.150,155.330
C06328=1066.017,166.379,420.177,172.844,29.147,155.329
C06329=1066.012,166.130,420.199,172.842,29.144,155.329
C06330=1066.006,165.881,420.221,172.841,29.141,155.328
C06331=1066.001,165.632,420.244,172.838,29.138,155.328
C06332=1065.995,165.383,420.266,172.837,29.136,155.328
C06333=1065.989,165.135,420.288,172.835,29.132,155.327
C06334=1065.984,164.885,420.310,172.833,29.130,155.327
C06335=1065.978,164.636,420.332,172.831,29.127,155.326
C06336=1065.973,164.388,420.354,172.829,29.124,155.326
C06337=1065.967,164.139,420.377,172.827,29.121,155.325
C06338=1065.962,163.889,420.399,172.826,29.118,155.325
C06339=1065.956,163.641,420.421,172.824,29.115,155.325
C06340=1065.950,163.392,420.443,172.822,29.112,155.324
C06341=1065.945,163.142,420.465,172.820,29.109,155.324
C06342=1065.939,162.894,420.487,172.818,29.106,155.323
C06343=1065.934,162.645,420.509,172.817,29.103,155.323
C06344=1065.928,162.395,420.531,172.814,29.100,155.322
C06345=1065.923,162.147,420.553,172.812,29.098,155.322
C06346=1065.917,161.898,420.576,172.811,29.095,155.321
C06347=1065.911,161.649,420.597,172.809,29.092,155.321
C06348=1065.906,161.400,420.619,172.808,29.089,155.321
C06349=1065.900,161.151,420.641,172.805,29.086,155.320
C06350=1065.895,160.902,420.664,172.803,29.083,155.320
C06351=1065.889,160.653,420.685,172.802,29.080,155.319
C06352=1065.882,160.404,420.707,172.800,29.077,155.319
C06353=1065.878,160.155,420.729,172.798,29.074,155.318
C06354=1065.871,159.906,420.750,172.796,29.072,155.318
C06355=1065.865,159.657,420.773,172.794,29.069,155.318
C06356=1065.860,159.408,420.795,172.793,29.066,155.317
C06357=1065.853,159.125,420.819,172.790,29.063,155.317
C06358=1065.846,158.842,420.844,172.788,29.060,155.316
C06359=1065.840,158.557,420.869,172.786,29.056,155.316
C06360=1065.834,158.275,420.893,172.784,29.053,155.315
C06361=1065.827,158.025,420.915,172.782,29.050,155.315
C06362=1065.821,157.777,420.937,172.780,29.048,155.314
C06363=1065.816,157.528,420.959,172.778,29.045,155.314
C06364=1065.810,157.279,420.980,172.777,29.042,155.314
C06365=1065.804,157.030,421.002,172.775,29.039,155.313
C06366=1065.799,156.781,421.024,172.773,29.036,155.313
C06367=1065.793,156.532,421.046,172.771,29.033,155.312
C06368=1065.787,156.283,421.067,172.769,29.030,155.312
C06369=1065.781,156.034,421.089,172.768,29.028,155.312
C06370=1065.776,155.784,421.111,172.766,29.025,155.311
C06371=1065.770,155.536,421.132,172.763,29.022,155.311
C06372=1065.764,155.287,421.154,172.762,29.019,155.310
C06373=1065.758,155.038,421.175,172.760,29.017,155.310
C06374=1065.752,154.789,421.197,172.758,29.014,155.309
C06375=1065.746,154.540,421.218,172.757,29.011,155.309
C06376=1065.741,154.291,421.240,172.755,29.008,155.309
C06377=1065.735,154.041,421.261,172.753,29.005,155.308
C06378=1065.730,153.793,421.282,172.751,29.002,155.308
C06379=1065.724,153.543,421.304,172.749,29.000,155.307
C06380=1065.718,153.295,421.325,172.748,28.997,155.307
C06381=1065.712,153.046,421.347,172.746,28.994,155.307
C06382=1065.706,152.796,421.368,172.744,28.991,155.306
C06383=1065.700,152.548,421.390,172.742,28.988,155.306
C06384=1065.695,152.298,421.412,172.740,28.986,155.305
C06385=1065.689,152.050,421.433,172.739,28.983,155.305
C06386=1065.683,151.800,421.454,172.737,28.980,155.304
C06387=1065.678,151.552,421.475,172.735,28.977,155.304
C06388=1065.672,151.302,421.497,172.733,28.974,155.304
C06389=1065.666,151.054,421.518,172.731,28.971,155.303
C06390=1065.660,150.805,421.540,172.730,28.969,155.303
C06391=1065.655,150.556,421.560,172.728,28.966,155.302
C06392=1065.649,150.306,421.582,172.726,28.963,155.302
C06393=1065.643,150.058,421.603,172.725,28.960,155.302
C06394=1065.637,149.809,421.625,172.722,28.958,155.301
C06395=1065.632,149.560,421.647,172.720,28.955,155.301
C06396=1065.626,149.310,421.668,172.719,28.952,155.300
C06397=1065.621,149.061,421.689,172.717,28.949,155.300
C06398=1065.614,148.812,421.711,172.716,28.946,155.299
C06399=1065.609,148.563,421.731,172.714,28.943,155.299
C06400=1065.603,148.314,421.753,172.712,28.941,155.299
C06401=1065.597,148.065,421.774,172.710,28.938,155.298
C06402=1065.591,147.816,421.796,172.708,28.935,155.298
C06403=1065.585,147.567,421.816,172.706,28.932,155.297
C06404=1065.579,147.318,421.837,172.705,28.930,155.297
C06405=1065.574,147.070,421.859,172.703,28.927,155.297
C06406=1065.568,146.820,421.880,172.702,28.924,155.296
C06407=1065.562,146.571,421.901,172.700,28.921,155.296
C06408=1065.556,146.322,421.922,172.697,28.918,155.295
C06409=1065.551,146.073,421.943,172.696,28.916,155.295
C06410=1065.545,145.824,421.965,172.694,28.913,155.295
C06411=1065.539,145.575,421.985,172.692,28.910,155.294
C06412=1065.532,145.326,422.006,172.691,28.908,155.294
C06413=1065.527,145.077,422.027,172.689,28.905,155.293
C06414=1065.521,144.827,422.048,172.688,28.902,155.293
C06415=1065.515,144.579,422.070,172.686,28.899,155.293
C06416=1065.510,144.329,422.091,172.683,28.896,155.292
C06417=1065.504,144.081,422.112,172.682,28.894,155.292
C06418=1065.498,143.832,422.132,172.680,28.891,155.291
C06419=1065.492,143.583,422.154,172.678,28.888,155.291
C06420=1065.487,143.334,422.174,172.677,28.885,155.290
C06421=1065.480,143.049,422.198,172.675,28.882,155.290
C06422=1065.474,142.766,422.222,172.673,28.879,155.290
C06423=1065.467,142.483,422.246,172.671,28.876,155.289
C06424=1065.460,142.199,422.270,172.669,28.872,155.289
C06425=1065.455,141.950,422.291,172.667,28.870,155.288
C06426=1065.448,141.701,422.312,172.665,28.867,155.288
C06427=1065.443,141.452,422.333,172.664,28.864,155.287
C06428=1065.437,141.202,422.353,172.662,28.861,155.287
C06429=1065.432,140.954,422.374,172.660,28.859,155.287
C06430=1065.426,140.704,422.395,172.659,28.856,155.286
C06431=1065.420,140.456,422.416,172.657,28.853,155.286
C06432=1065.414,140.206,422.437,172.655,28.850,155.285
C06433=1065.409,139.957,422.457,172.653,28.847,155.285
C06434=1065.403,139.708,422.479,172.651,28.844,155.284
C06435=1065.396,139.459,422.499,172.650,28.842,155.284
C06436=1065.391,139.210,422.520,172.648,28.839,155.284
C06437=1065.386,138.961,422.541,172.647,28.836,155.283
C06438=1065.379,138.712,422.561,172.645,28.833,155.283
C06439=1065.373,138.463,422.582,172.643,28.831,155.282
C06440=1065.368,138.213,422.603,172.642,28.828,155.282
C06441=1065.362,137.965,422.623,172.640,28.825,155.282
C06442=1065.356,137.715,422.644,172.638,28.822,155.281
C06443=1065.350,137.466,422.666,172.636,28.820,155.281
C06444=1065.344,137.217,422.685,172.634,28.817,155.280
C06445=1065.339,136.968,422.706,172.633,28.814,155.280
C06446=1065.333,136.719,422.728,172.631,28.811,155.280
C06447=1065.327,136.470,422.748,172.629,28.809,155.279
C06448=1065.321,136.221,422.768,172.628,28.806,155.279
C06449=1065.315,135.972,422.789,172.626,28.803,155.278
C06450=1065.309,135.723,422.810,172.624,28.800,155.278
C06451=1065.304,135.474,422.830,172.623,28.798,155.278
C06452=1065.297,135.225,422.851,172.621,28.795,155.277
C06453=1065.292,134.975,422.871,172.620,28.792,155.277
C06454=1065.286,134.727,422.891,172.618,28.789,155.276
C06455=1065.281,134.478,422.912,172.616,28.787,155.276
C06456=1065.274,134.229,422.933,172.614,28.784,155.276
C06457=1065.269,133.979,422.953,172.612,28.781,155.275
C06458=1065.264,133.730,422.974,172.611,28.778,155.275
C06459=1065.257,133.481,422.994,172.609,28.776,155.274
C06460=1065.252,133.232,423.015,172.607,28.773,155.274
C06461=1065.246,132.983,423.035,172.606,28.770,155.274
C06462=1065.240,132.734,423.056,172.604,28.767,155.273
C06463=1065.234,132.485,423.076,172.602,28.765,155.273
C06464=1065.228,132.236,423.097,172.601,28.762,155.272
C06465=1065.223,131.987,423.117,172.599,28.759,155.272
C06466=1065.217,131.738,423.137,172.598,28.756,155.272
C06467=1065.210,131.488,423.158,172.596,28.754,155.271
C06468=1065.205,131.239,423.178,172.594,28.751,155.271
C06469=1065.199,130.990,423.198,172.593,28.748,155.270
C06470=1065.193,130.741,423.219,172.591,28.745,155.270
C06471=1065.187,130.492,423.239,172.590,28.743,155.269
C06472=1065.181,130.243,423.259,172.587,28.740,155.269
C06473=1065.175,129.994,423.279,172.585,28.738,155.269
C06474=1065.169,129.744,423.300,172.584,28.735,155.268
C06475=1065.163,129.495,423.320,172.582,28.732,155.268
C06476=1065.158,129.247,423.340,172.580,28.729,155.268
C06477=1065.151,128.997,423.360,172.579,28.727,155.267
C06478=1065.146,128.748,423.381,172.577,28.724,155.267
C06479=1065.140,128.499,423.401,172.576,28.721,155.266
C06480=1065.134,128.250,423.421,172.574,28.718,155.266
C06481=1065.128,128.001,423.442,172.572,28.716,155.266
C06482=1065.122,127.752,423.462,172.571,28.713,155.265
C06483=1065.116,127.503,423.481,172.569,28.710,155.265
C06484=1065.110,127.254,423.501,172.567,28.707,155.264
C06485=1065.103,126.969,423.525,172.566,28.705,155.264
C06486=1065.097,126.686,423.547,172.563,28.701,155.263
C06487=1065.090,126.403,423.570,172.562,28.698,155.263
C06488=1065.084,126.118,423.593,172.560,28.695,155.263
C06489=1065.078,125.869,423.613,172.559,28.692,155.262
C06490=1065.072,125.620,423.633,172.557,28.690,155.262
C06491=1065.066,125.372,423.653,172.555,28.687,155.261
C06492=1065.060,125.121,423.673,172.553,28.684,155.261
C06493=1065.054,124.872,423.693,172.551,28.682,155.261
C06494=1065.048,124.624,423.713,172.550,28.679,155.260
C06495=1065.042,124.375,423.733,172.548,28.676,155.260
C06496=1065.037,124.126,423.754,172.546,28.673,155.259
C06497=1065.031,123.877,423.774,172.545,28.671,155.259
C06498=1065.025,123.627,423.793,172.543,28.668,155.259
C06499=1065.019,123.378,423.813,172.541,28.665,155.258
C06500=1065.013,123.129,423.834,172.540,28.662,155.258
C06501=1065.007,122.880,423.854,172.538,28.660,155.257
C06502=1065.002,122.631,423.873,172.537,28.657,155.257
C06503=1064.996,122.382,423.893,172.535,28.654,155.257
C06504=1064.990,122.133,423.913,172.533,28.651,155.256
C06505=1064.984,121.884,423.934,172.532,28.649,155.256
C06506=1064.978,121.634,423.953,172.530,28.646,155.255
C06507=1064.972,121.385,423.973,172.529,28.643,155.255
C06508=1064.966,121.136,423.993,172.527,28.640,155.255
C06509=1064.961,120.886,424.013,172.525,28.638,155.254
C06510=1064.955,120.637,424.033,172.524,28.635,155.254
C06511=1064.949,120.389,424.053,172.522,28.632,155.253
C06512=1064.943,120.139,424.072,172.521,28.629,155.253
C06513=1064.937,119.890,424.092,172.519,28.627,155.253
C06514=1064.932,119.641,424.113,172.517,28.624,155.252
C06515=1064.927,119.392,424.132,172.516,28.621,155.252
C06516=1064.921,119.143,424.152,172.514,28.618,155.251
C06517=1064.915,118.894,424.171,172.513,28.616,155.251
C06518=1064.909,118.645,424.191,172.511,28.613,155.251
C06519=1064.904,118.396,424.212,172.509,28.610,155.250
C06520=1064.897,118.146,424.231,172.508,28.607,155.250
C06521=1064.891,117.897,424.251,172.506,28.605,155.249
C06522=1064.886,117.647,424.270,172.505,28.602,155.249
C06523=1064.880,117.398,424.290,172.503,28.599,155.248
C06524=1064.874,117.150,424.310,172.501,28.596,155.248
C06525=1064.869,116.900,424.330,172.500,28.593,155.248
C06526=1064.863,116.651,424.350,172.498,28.590,155.247
C06527=1064.857,116.402,424.369,172.497,28.588,155.247
C06528=1064.851,116.153,424.389,172.495,28.585,155.246
C06529=1064.845,115.903,424.409,172.493,28.582,155.246
C06530=1064.839,115.655,424.429,172.492,28.579,155.246
C06531=1064.834,115.405,424.448,172.490,28.577,155.245
C06532=1064.828,115.156,424.468,172.489,28.574,155.245
C06533=1064.823,114.907,424.488,172.487,28.571,155.244
C06534=1064.817,114.658,424.508,172.485,28.568,155.244
C06535=1064.812,114.409,424.526,172.485,28.566,155.244
C06536=1064.806,114.160,424.546,172.483,28.563,155.243
C06537=1064.800,113.911,424.566,172.482,28.560,155.243
C06538=1064.794,113.661,424.585,172.480,28.558,155.242
C06539=1064.788,113.412,424.605,172.478,28.555,155.242
C06540=1064.782,113.162,424.624,172.477,28.552,155.242
C06541=1064.776,112.914,424.644,172.475,28.549,155.241
C06542=1064.770,112.664,424.664,172.474,28.547,155.241
C06543=1064.765,112.415,424.683,172.472,28.544,155.240
C06544=1064.759,112.166,424.703,172.470,28.541,155.240
C06545=1064.754,111.917,424.722,172.469,28.538,155.240
C06546=1064.748,111.668,424.741,172.467,28.536,155.239
C06547=1064.742,111.419,424.761,172.466,28.533,155.239
C06548=1064.735,111.170,424.780,172.464,28.530,155.238
C06549=1064.728,110.885,424.802,172.462,28.527,155.238
C06550=1064.722,110.602,424.825,172.460,28.524,155.237
C06551=1064.715,110.318,424.846,172.458,28.521,155.237
C06552=1064.708,110.034,424.868,172.457,28.518,155.236
C06553=1064.703,109.785,424.887,172.455,28.515,155.236
C06554=1064.697,109.536,424.907,172.454,28.513,155.236
C06555=1064.691,109.287,424.926,172.452,28.510,155.235
C06556=1064.685,109.037,424.946,172.450,28.507,155.235
C06557=1064.679,108.788,424.964,172.449,28.504,155.235
C06558=1064.673,108.539,424.984,172.447,28.502,155.234
C06559=1064.667,108.290,425.004,172.446,28.499,155.234
C06560=1064.661,108.040,425.023,172.444,28.496,155.233
C06561=1064.655,107.791,425.041,172.442,28.493,155.233
C06562=1064.649,107.542,425.061,172.441,28.491,155.233
C06563=1064.643,107.293,425.081,172.439,28.488,155.232
C06564=1064.638,107.044,425.100,172.438,28.485,155.232
C06565=1064.632,106.794,425.119,172.436,28.482,155.231
C06566=1064.626,106.546,425.137,172.434,28.480,155.231
C06567=1064.620,106.296,425.157,172.433,28.477,155.231
C06568=1064.615,106.047,425.176,172.431,28.475,155.230
C06569=1064.609,105.798,425.196,172.430,28.472,155.230
C06570=1064.602,105.549,425.214,172.429,28.469,155.229
C06571=1064.597,105.299,425.234,172.427,28.467,155.229
C06572=1064.591,105.050,425.253,172.426,28.464,155.229
C06573=1064.585,104.801,425.272,172.424,28.461,155.228
C06574=1064.579,104.551,425.291,172.423,28.458,155.228
C06575=1064.574,104.303,425.310,172.421,28.455,155.227
C06576=1064.568,104.053,425.329,172.419,28.453,155.227
C06577=1064.561,103.805,425.348,172.418,28.450,155.227
C06578=1064.556,103.555,425.368,172.416,28.447,155.226
C06579=1064.550,103.306,425.387,172.415,28.444,155.226
C06580=1064.544,103.056,425.406,172.413,28.442,155.225
C06581=1064.538,102.807,425.425,172.411,28.439,155.225
C06582=1064.533,102.559,425.444,172.410,28.436,155.225
C06583=1064.527,102.309,425.463,172.408,28.433,155.224
C06584=1064.521,102.060,425.481,172.407,28.431,155.224
C06585=1064.515,101.811,425.501,172.405,28.428,155.223
C06586=1064.509,101.561,425.520,172.404,28.425,155.223
C06587=1064.503,101.312,425.539,172.403,28.423,155.223
C06588=1064.498,101.063,425.557,172.401,28.420,155.222
C06589=1064.492,100.814,425.577,172.400,28.417,155.222
C06590=1064.486,100.565,425.595,172.398,28.414,155.221
C06591=1064.480,100.315,425.615,172.396,28.411,155.221
C06592=1064.473,100.066,425.633,172.395,28.409,155.221
C06593=1064.468,99.817,425.653,172.393,28.407,155.220
C06594=1064.461,99.568,425.671,172.392,28.404,155.220
C06595=1064.457,99.318,425.689,172.390,28.401,155.219
C06596=1064.450,99.069,425.708,172.388,28.398,155.219
C06597=1064.444,98.820,425.727,172.387,28.395,155.219
C06598=1064.438,98.571,425.746,172.385,28.393,155.218
C06599=1064.432,98.321,425.765,172.384,28.390,155.218
C06600=1064.426,98.073,425.783,172.382,28.387,155.217
C06601=1064.421,97.823,425.803,172.382,28.385,155.217
C06602=1064.414,97.574,425.821,172.380,28.382,155.217
C06603=1064.409,97.325,425.841,172.378,28.380,155.216
C06604=1064.403,97.075,425.858,172.377,28.377,155.216
C06605=1064.397,96.826,425.878,172.375,28.374,155.216
C06606=1064.391,96.577,425.896,172.374,28.371,155.215
C06607=1064.385,96.328,425.915,172.372,28.369,155.215
C06608=1064.379,96.079,425.934,172.370,28.366,155.214
C06609=1064.374,95.829,425.952,172.369,28.363,155.214
C06610=1064.368,95.580,425.971,172.367,28.360,155.214
C06611=1064.361,95.331,425.989,172.366,28.357,155.213
C06612=1064.356,95.082,426.009,172.364,28.355,155.213
C06613=1064.349,94.798,426.030,172.362,28.352,155.212
C06614=1064.342,94.513,426.051,172.361,28.349,155.212
C06615=1064.336,94.230,426.072,172.359,28.346,155.211
C06616=1064.329,93.946,426.093,172.358,28.342,155.211
C06617=1064.323,93.697,426.112,172.356,28.340,155.211
C06618=1064.317,93.448,426.131,172.355,28.337,155.210
C06619=1064.311,93.199,426.149,172.353,28.334,155.210
C06620=1064.306,92.949,426.168,172.352,28.331,155.209
C06621=1064.299,92.700,426.186,172.350,28.329,155.209
C06622=1064.294,92.451,426.205,172.348,28.326,155.209
C06623=1064.288,92.202,426.223,172.347,28.324,155.208
C06624=1064.282,91.952,426.242,172.345,28.321,155.208
C06625=1064.276,91.703,426.261,172.344,28.318,155.207
C06626=1064.270,91.454,426.278,172.342,28.315,155.207
C06627=1064.265,91.205,426.298,172.341,28.313,155.207
C06628=1064.258,90.955,426.316,172.340,28.310,155.206
C06629=1064.254,90.706,426.335,172.338,28.307,155.206
C06630=1064.247,90.457,426.353,172.337,28.304,155.205
C06631=1064.241,90.207,426.371,172.335,28.302,155.205
C06632=1064.235,89.958,426.390,172.333,28.299,155.205
C06633=1064.229,89.710,426.408,172.332,28.296,155.204
C06634=1064.223,89.460,426.427,172.330,28.293,155.204
C06635=1064.217,89.210,426.445,172.329,28.291,155.204
C06636=1064.211,88.961,426.463,172.327,28.288,155.203
C06637=1064.205,88.712,426.481,172.326,28.286,155.203
C06638=1064.199,88.463,426.499,172.325,28.283,155.202
C06639=1064.193,88.213,426.519,172.323,28.280,155.202
C06640=1064.187,87.965,426.537,172.322,28.278,155.201
C06641=1064.181,87.715,426.555,172.320,28.275,155.201
C06642=1064.175,87.466,426.573,172.319,28.273,155.201
C06643=1064.169,87.217,426.591,172.317,28.270,155.200
C06644=1064.164,86.967,426.610,172.315,28.267,155.200
C06645=1064.157,86.718,426.628,172.314,28.264,155.200
C06646=1064.152,86.469,426.647,172.312,28.261,155.199
C06647=1064.146,86.219,426.664,172.311,28.259,155.199
C06648=1064.139,85.970,426.682,172.309,28.256,155.198
C06649=1064.134,85.721,426.701,172.308,28.253,155.198
C06650=1064.127,85.472,426.719,172.307,28.251,155.198
C06651=1064.122,85.222,426.738,172.305,28.248,155.197
C06652=1064.116,84.973,426.755,172.304,28.246,155.197
C06653=1064.110,84.724,426.774,172.302,28.243,155.197
C06654=1064.104,84.474,426.792,172.301,28.240,155.196
C06655=1064.098,84.225,426.810,172.299,28.237,155.196
C06656=1064.092,83.976,426.828,172.297,28.234,155.195
C06657=1064.087,83.727,426.846,172.296,28.232,155.195
C06658=1064.081,83.478,426.865,172.295,28.229,155.194
C06659=1064.074,83.228,426.883,172.294,28.226,155.194
C06660=1064.069,82.979,426.901,172.292,28.224,155.194
C06661=1064.063,82.730,426.919,172.291,28.221,155.193
C06662=1064.057,82.481,426.937,172.289,28.219,155.193
C06663=1064.051,82.231,426.955,172.287,28.216,155.193
C06664=1064.044,81.982,426.973,172.286,28.213,155.192
C06665=1064.040,81.732,426.991,172.284,28.210,155.192
C06666=1064.034,81.483,427.009,172.283,28.207,155.191
C06667=1064.028,81.234,427.028,172.281,28.205,155.191
C06668=1064.022,80.985,427.046,172.280,28.202,155.191
C06669=1064.016,80.736,427.063,172.279,28.199,155.190
C06670=1064.010,80.486,427.082,172.277,28.197,155.190
C06671=1064.004,80.237,427.099,172.276,28.194,155.189
C06672=1063.998,79.988,427.117,172.274,28.191,155.189
C06673=1063.993,79.739,427.135,172.273,28.188,155.189
C06674=1063.987,79.489,427.154,172.271,28.185,155.188
C06675=1063.981,79.239,427.172,172.269,28.183,155.188
C06676=1063.975,78.990,427.190,172.269,28.180,155.187
C06677=1063.967,78.707,427.210,172.266,28.177,155.187
C06678=1063.961,78.423,427.230,172.265,28.174,155.187
C06679=1063.954,78.139,427.251,172.263,28.171,155.186
C06680=1063.948,77.855,427.271,172.262,28.168,155.186
C06681=1063.942,77.606,427.290,172.260,28.165,155.185
C06682=1063.936,77.357,427.307,172.259,28.163,155.185
C06683=1063.930,77.107,427.325,172.257,28.160,155.184
C06684=1063.924,76.858,427.342,172.255,28.157,155.184
C06685=1063.918,76.609,427.360,172.255,28.154,155.184
C06686=1063.912,76.360,427.378,172.253,28.152,155.183
C06687=1063.906,76.110,427.396,172.252,28.149,155.183
C06688=1063.900,75.861,427.414,172.250,28.147,155.183
C06689=1063.894,75.612,427.432,172.248,28.144,155.182
C06690=1063.888,75.362,427.450,172.247,28.141,155.182
C06691=1063.883,75.113,427.467,172.245,28.138,155.181
C06692=1063.876,74.863,427.485,172.244,28.135,155.181
C06693=1063.870,74.614,427.502,172.242,28.133,155.181
C06694=1063.864,74.365,427.520,172.242,28.131,155.180
C06695=1063.859,74.116,427.538,172.240,28.128,155.180
C06696=1063.853,73.866,427.556,172.238,28.125,155.179
C06697=1063.847,73.617,427.573,172.237,28.122,155.179
C06698=1063.841,73.367,427.591,172.235,28.120,155.179
C06699=1063.834,73.119,427.609,172.234,28.117,155.178
C06700=1063.828,72.869,427.627,172.232,28.114,155.178
C06701=1063.823,72.620,427.644,172.231,28.111,155.177
C06702=1063.817,72.371,427.662,172.230,28.109,155.177
C06703=1063.811,72.121,427.680,172.228,28.106,155.177
C06704=1063.806,71.872,427.697,172.227,28.104,155.176
C06705=1063.799,71.623,427.715,172.225,28.101,155.176
C06706=1063.793,71.374,427.732,172.224,28.098,155.176
C06707=1063.787,71.124,427.750,172.222,28.095,155.175
C06708=1063.782,70.875,427.767,172.221,28.092,155.175
C06709=1063.776,70.625,427.785,172.219,28.090,155.174
C06710=1063.769,70.376,427.802,172.218,28.088,155.174
C06711=1063.764,70.127,427.819,172.217,28.085,155.174
C06712=1063.758,69.877,427.837,172.215,28.082,155.173
C06713=1063.752,69.628,427.855,172.214,28.079,155.173
C06714=1063.745,69.379,427.872,172.212,28.077,155.172
C06715=1063.740,69.130,427.890,172.211,28.074,155.172
C06716=1063.734,68.880,427.908,172.209,28.071,155.172
C06717=1063.728,68.631,427.925,172.207,28.069,155.171
C06718=1063.721,68.382,427.943,172.206,28.066,155.171
C06719=1063.716,68.133,427.960,172.205,28.063,155.171
C06720=1063.711,67.883,427.977,172.204,28.061,155.170
C06721=1063.704,67.633,427.994,172.202,28.058,155.170
C06722=1063.698,67.384,428.012,172.201,28.055,155.169
C06723=1063.692,67.135,428.030,172.199,28.052,155.169
C06724=1063.686,66.886,428.047,172.197,28.050,155.169
C06725=1063.680,66.637,428.065,172.196,28.047,155.168
C06726=1063.674,66.387,428.081,172.195,28.045,155.168
C06727=1063.668,66.138,428.099,172.194,28.042,155.167
C06728=1063.662,65.888,428.117,172.192,28.039,155.167
C06729=1063.656,65.639,428.134,172.191,28.036,155.167
C06730=1063.650,65.390,428.151,172.189,28.034,155.166
C06731=1063.645,65.140,428.168,172.187,28.031,155.166
C06732=1063.638,64.891,428.185,172.186,28.028,155.166
C06733=1063.632,64.641,428.203,172.184,28.026,155.165
C06734=1063.626,64.393,428.220,172.184,28.023,155.165
C06735=1063.621,64.143,428.237,172.182,28.020,155.164
C06736=1063.614,63.894,428.254,172.180,28.018,155.164
C06737=1063.608,63.645,428.272,172.179,28.015,155.164
C06738=1063.602,63.395,428.289,172.177,28.012,155.163
C06739=1063.596,63.145,428.306,172.176,28.010,155.163
C06740=1063.590,62.897,428.323,172.174,28.007,155.163
C06741=1063.583,62.612,428.343,172.173,28.005,155.162
C06742=1063.576,62.329,428.362,172.171,28.001,155.162
C06743=1063.568,62.045,428.382,172.170,27.998,155.161
C06744=1063.562,61.760,428.401,172.168,27.996,155.161
C06745=1063.556,61.511,428.418,172.167,27.993,155.161
C06746=1063.550,61.262,428.435,172.165,27.990,155.160
C06747=1063.544,61.012,428.452,172.163,27.988,155.160
C06748=1063.537,60.763,428.470,172.162,27.985,155.159
C06749=1063.531,60.514,428.487,172.160,27.982,155.159
C06750=1063.526,60.265,428.503,172.159,27.979,155.159
C06751=1063.519,60.015,428.521,172.158,27.977,155.158
C06752=1063.513,59.766,428.537,172.156,27.975,155.158
C06753=1063.508,59.517,428.555,172.155,27.972,155.158
C06754=1063.501,59.267,428.572,172.153,27.969,155.157
C06755=1063.496,59.018,428.589,172.152,27.967,155.157
C06756=1063.489,58.769,428.606,172.150,27.964,155.157
C06757=1063.483,58.519,428.622,172.149,27.961,155.156
C06758=1063.477,58.270,428.640,172.148,27.959,155.156
C06759=1063.471,58.020,428.656,172.146,27.956,155.155
C06760=1063.464,57.771,428.674,172.145,27.954,155.155
C06761=1063.459,57.521,428.690,172.143,27.951,155.155
C06762=1063.453,57.273,428.707,172.142,27.948,155.154
C06763=1063.446,57.023,428.724,172.140,27.946,155.154
C06764=1063.441,56.774,428.742,172.139,27.943,155.154
C06765=1063.435,56.524,428.758,172.137,27.940,155.153
C06766=1063.429,56.275,428.775,172.136,27.938,155.153
C06767=1063.423,56.025,428.792,172.135,27.935,155.152
C06768=1063.417,55.776,428.809,172.133,27.933,155.152
C06769=1063.411,55.527,428.825,172.132,27.930,155.152
C06770=1063.405,55.277,428.843,172.130,27.927,155.151
C06771=1063.399,55.028,428.859,172.129,27.924,155.151
C06772=1063.393,54.779,428.876,172.127,27.922,155.151
C06773=1063.387,54.530,428.893,172.125,27.919,155.150
C06774=1063.381,54.279,428.910,172.125,27.917,155.150
C06775=1063.374,54.031,428.927,172.123,27.914,155.149
C06776=1063.369,53.781,428.944,172.122,27.912,155.149
C06777=1063.363,53.532,428.961,172.120,27.909,155.149
C06778=1063.357,53.283,428.977,172.119,27.906,155.148
C06779=1063.351,53.033,428.994,172.117,27.903,155.148
C06780=1063.345,52.784,429.011,172.116,27.900,155.148
C06781=1063.339,52.535,429.027,172.115,27.898,155.147
C06782=1063.333,52.285,429.044,172.113,27.896,155.147
C06783=1063.327,52.035,429.062,172.112,27.893,155.146
C06784=1063.321,51.786,429.078,172.110,27.890,155.146
C06785=1063.315,51.537,429.094,172.109,27.887,155.146
C06786=1063.309,51.288,429.112,172.107,27.885,155.145
C06787=1063.303,51.038,429.128,172.106,27.882,155.145
C06788=1063.298,50.789,429.144,172.105,27.879,155.145
C06789=1063.291,50.540,429.162,172.103,27.877,155.144
C06790=1063.285,50.290,429.178,172.102,27.874,155.144
C06791=1063.279,50.041,429.195,172.100,27.872,155.143
C06792=1063.273,49.792,429.212,172.099,27.869,155.143
C06793=1063.268,49.542,429.228,172.097,27.866,155.143
C06794=1063.262,49.293,429.245,172.096,27.863,155.142
C06795=1063.256,49.043,429.261,172.094,27.860,155.142
C06796=1063.249,48.794,429.278,172.093,27.858,155.142
C06797=1063.244,48.544,429.295,172.092,27.856,155.141
C06798=1063.238,48.295,429.311,172.090,27.853,155.141
C06799=1063.232,48.046,429.328,172.089,27.850,155.140
C06800=1063.226,47.796,429.344,172.087,27.847,155.140
C06801=1063.221,47.547,429.361,172.086,27.844,155.140
C06802=1063.215,47.298,429.378,172.084,27.842,155.139
C06803=1063.208,47.048,429.394,172.084,27.840,155.139
C06804=1063.202,46.799,429.411,172.082,27.837,155.139
C06805=1063.196,46.514,429.429,172.080,27.834,155.138
C06806=1063.189,46.231,429.449,172.078,27.830,155.138
C06807=1063.182,45.947,429.467,172.077,27.827,155.137
C06808=1063.175,45.662,429.486,172.075,27.825,155.137
C06809=1063.170,45.412,429.503,172.073,27.822,155.136
C06810=1063.164,45.163,429.519,172.073,27.819,155.136
C06811=1063.158,44.913,429.536,172.071,27.816,155.136
C06812=1063.152,44.665,429.553,172.070,27.814,155.135
C06813=1063.146,44.415,429.569,172.068,27.811,155.135
C06814=1063.141,44.166,429.586,172.067,27.809,155.135
C06815=1063.135,43.916,429.602,172.065,27.806,155.134
C06816=1063.129,43.667,429.618,172.064,27.803,155.134
C06817=1063.123,43.418,429.634,172.063,27.800,155.133
C06818=1063.117,43.168,429.651,172.062,27.798,155.133
C06819=1063.111,42.919,429.667,172.060,27.795,155.133
C06820=1063.105,42.670,429.683,172.058,27.793,155.132
C06821=1063.099,42.420,429.700,172.057,27.790,155.132
C06822=1063.093,42.170,429.716,172.055,27.787,155.132
C06823=1063.087,41.921,429.732,172.054,27.785,155.131
C06824=1063.081,41.671,429.749,172.052,27.782,155.131
C06825=1063.075,41.422,429.765,172.052,27.779,155.130
C06826=1063.069,41.173,429.781,172.050,27.777,155.130
C06827=1063.063,40.923,429.797,172.048,27.774,155.130
C06828=1063.057,40.674,429.814,172.047,27.771,155.129
C06829=1063.051,40.425,429.830,172.045,27.769,155.129
C06830=1063.045,40.175,429.846,172.044,27.766,155.129
C06831=1063.039,39.926,429.862,172.042,27.764,155.128
C06832=1063.033,39.677,429.879,172.042,27.761,155.128
C06833=1063.027,39.427,429.895,172.040,27.759,155.128
C06834=1063.021,39.178,429.911,172.038,27.756,155.127
C06835=1063.015,38.929,429.927,172.037,27.753,155.127
C06836=1063.009,38.679,429.944,172.035,27.750,155.126
C06837=1063.003,38.430,429.960,172.034,27.748,155.126
C06838=1062.997,38.181,429.976,172.032,27.745,155.126
C06839=1062.992,37.931,429.992,172.031,27.742,155.125
C06840=1062.986,37.681,430.008,172.030,27.740,155.125
C06841=1062.980,37.432,430.024,172.029,27.738,155.125
C06842=1062.973,37.182,430.040,172.027,27.735,155.124
C06843=1062.967,36.933,430.057,172.025,27.733,155.124
C06844=1062.961,36.683,430.073,172.024,27.730,155.124
C06845=1062.955,36.434,430.089,172.022,27.727,155.123
C06846=1062.949,36.184,430.105,172.021,27.725,155.123
C06847=1062.942,35.935,430.120,172.020,27.722,155.122
C06848=1062.936,35.686,430.136,172.019,27.719,155.122
C06849=1062.930,35.436,430.153,172.017,27.717,155.122
C06850=1062.924,35.187,430.169,172.016,27.714,155.121
C06851=1062.918,34.937,430.184,172.014,27.712,155.121
C06852=1062.912,34.688,430.200,172.012,27.709,155.121
C06853=1062.906,34.439,430.216,172.011,27.706,155.120
C06854=1062.900,34.189,430.233,172.009,27.704,155.120
C06855=1062.894,33.940,430.249,172.009,27.701,155.120
C06856=1062.888,33.690,430.264,172.007,27.699,155.119
C06857=1062.882,33.441,430.280,172.006,27.696,155.119
C06858=1062.876,33.192,430.296,172.004,27.694,155.119
C06859=1062.870,32.942,430.313,172.002,27.691,155.118
C06860=1062.864,32.693,430.328,172.001,27.689,155.118
C06861=1062.858,32.443,430.344,171.999,27.686,155.118
C06862=1062.852,32.195,430.360,171.998,27.683,155.117
C06863=1062.847,31.945,430.375,171.997,27.681,155.117
C06864=1062.840,31.696,430.391,171.996,27.678,155.116
C06865=1062.834,31.446,430.407,171.994,27.676,155.116
C06866=1062.828,31.196,430.423,171.993,27.673,155.116
C06867=1062.822,30.947,430.439,171.991,27.670,155.115
C06868=1062.816,30.698,430.455,171.989,27.668,155.115
C06869=1062.806,30.302,430.480,171.987,27.664,155.115
C06870=1062.797,29.906,430.505,171.985,27.659,155.114
C06871=1062.788,29.511,430.530,171.983,27.655,155.113
C06872=1062.778,29.115,430.555,171.980,27.651,155.113
C06873=1062.769,28.728,430.579,171.978,27.647,155.112
C06874=1062.759,28.340,430.604,171.977,27.643,155.112
C06875=1062.750,27.953,430.628,171.974,27.640,155.111
C06876=1062.741,27.566,430.652,171.972,27.635,155.111
C06877=1062.735,27.316,430.668,171.970,27.633,155.110
C06878=1062.728,27.067,430.684,171.969,27.630,155.110
C06879=1062.723,26.817,430.699,171.967,27.627,155.110
C06880=1062.716,26.568,430.715,171.966,27.625,155.109
C06881=1062.710,26.318,430.730,171.964,27.622,155.109
C06882=1062.704,26.068,430.747,171.963,27.620,155.109
C06883=1062.698,25.819,430.761,171.962,27.618,155.108
C06884=1062.692,25.569,430.778,171.960,27.615,155.108
C06885=1062.686,25.320,430.793,171.959,27.612,155.108
C06886=1062.680,25.071,430.809,171.957,27.610,155.107
C06887=1062.674,24.821,430.823,171.956,27.607,155.107
C06888=1062.668,24.572,430.840,171.954,27.605,155.107
C06889=1062.662,24.322,430.855,171.953,27.602,155.106
C06890=1062.656,24.073,430.871,171.951,27.599,155.106
C06891=1062.649,23.823,430.886,171.950,27.597,155.106
C06892=1062.643,23.574,430.902,171.949,27.595,155.105
C06893=1062.637,23.325,430.917,171.947,27.592,155.105
C06894=1062.632,23.075,430.932,171.946,27.590,155.104
C06895=1062.625,22.826,430.948,171.944,27.587,155.104
C06896=1062.620,22.576,430.963,171.943,27.584,155.104
C06897=1062.613,22.327,430.979,171.941,27.582,155.103
C06898=1062.607,22.077,430.995,171.940,27.579,155.103
C06899=1062.601,21.828,431.009,171.939,27.577,155.103
C06900=1062.595,21.579,431.026,171.937,27.575,155.102
C06901=1062.589,21.329,431.040,171.936,27.572,155.102
C06902=1062.583,21.079,431.056,171.934,27.569,155.102
C06903=1062.577,20.830,431.072,171.933,27.567,155.101
C06904=1062.572,20.581,431.087,171.931,27.564,155.101
C06905=1062.565,20.331,431.102,171.930,27.562,155.101
C06906=1062.559,20.082,431.118,171.928,27.559,155.100
C06907=1062.553,19.832,431.133,171.928,27.557,155.100
C06908=1062.547,19.582,431.148,171.926,27.554,155.100
C06909=1062.541,19.334,431.164,171.924,27.552,155.099
C06910=1062.535,19.084,431.179,171.923,27.549,155.099
C06911=1062.528,18.834,431.194,171.921,27.547,155.099
C06912=1062.523,18.585,431.209,171.920,27.544,155.098
C06913=1062.516,18.335,431.225,171.918,27.541,155.098
C06914=1062.511,18.086,431.240,171.917,27.539,155.098
C06915=1062.505,17.837,431.255,171.915,27.536,155.097
C06916=1062.498,17.587,431.270,171.914,27.534,155.097
C06917=1062.492,17.338,431.286,171.913,27.532,155.097
C06918=1062.486,17.088,431.301,171.911,27.529,155.096
C06919=1062.480,16.839,431.316,171.910,27.526,155.096
C06920=1062.475,16.589,431.331,171.908,27.524,155.096
C06921=1062.468,16.340,431.347,171.907,27.521,155.095
C06922=1062.461,16.090,431.362,171.905,27.519,155.095
C06923=1062.456,15.841,431.377,171.904,27.516,155.095
C06924=1062.450,15.591,431.392,171.902,27.514,155.094
C06925=1062.444,15.342,431.407,171.901,27.511,155.094
C06926=1062.439,15.092,431.422,171.900,27.509,155.094
C06927=1062.432,14.843,431.438,171.898,27.506,155.093
C06928=1062.426,14.594,431.453,171.897,27.504,155.093
C06929=1062.419,14.311,431.470,171.895,27.501,155.093
C06930=1062.412,14.028,431.486,171.894,27.498,155.092
C06931=1062.405,13.745,431.503,171.891,27.495,155.092
C06932=1062.398,13.462,431.521,171.890,27.492,155.092
C06933=1062.392,13.212,431.536,171.888,27.490,155.091
C06934=1062.386,12.962,431.551,171.887,27.488,155.091
C06935=1062.380,12.714,431.566,171.886,27.485,155.091
C06936=1062.373,12.464,431.581,171.884,27.483,155.090
C06937=1062.367,12.214,431.596,171.883,27.481,155.090
C06938=1062.361,11.965,431.610,171.881,27.478,155.090
C06939=1062.355,11.716,431.625,171.880,27.476,155.089
C06940=1062.349,11.466,431.641,171.878,27.473,155.089
C06941=1062.343,11.216,431.656,171.877,27.471,155.089
C06942=1062.337,10.967,431.670,171.875,27.468,155.088
C06943=1062.331,10.717,431.685,171.873,27.466,155.088
C06944=1062.324,10.468,431.700,171.873,27.464,155.088
C06945=1062.318,10.218,431.715,171.871,27.461,155.087
C06946=1062.312,9.969,431.730,171.870,27.458,155.087
C06947=1062.306,9.719,431.744,171.868,27.456,155.087
C06948=1062.299,9.470,431.759,171.867,27.454,155.087
C06949=1062.294,9.221,431.774,171.865,27.451,155.086
C06950=1062.287,8.971,431.789,171.863,27.449,155.086
C06951=1062.282,8.721,431.804,171.862,27.447,155.086
C06952=1062.276,8.472,431.819,171.860,27.444,155.085
C06953=1062.269,8.223,431.834,171.859,27.441,155.085
C06954=1062.263,7.973,431.849,171.858,27.439,155.085
C06955=1062.257,7.724,431.864,171.857,27.437,155.084
C06956=1062.251,7.474,431.878,171.855,27.434,155.084
C06957=1062.245,7.225,431.893,171.854,27.431,155.084
C06958=1062.239,6.976,431.908,171.852,27.429,155.083
C06959=1062.232,6.726,431.923,171.850,27.427,155.083
C06960=1062.226,6.476,431.937,171.849,27.424,155.083
C06961=1062.220,6.227,431.952,171.847,27.422,155.082
C06962=1062.214,5.977,431.967,171.846,27.420,155.082
C06963=1062.208,5.728,431.981,171.844,27.417,155.082
C06964=1062.202,5.479,431.996,171.843,27.414,155.081
C06965=1062.196,5.229,432.011,171.842,27.412,155.081
C06966=1062.190,4.980,432.026,171.840,27.410,155.081
C06967=1062.184,4.730,432.040,171.839,27.407,155.081
C06968=1062.179,4.480,432.055,171.837,27.405,155.080
C06969=1062.172,4.231,432.070,171.836,27.402,155.080
C06970=1062.166,3.981,432.085,171.834,27.400,155.080
C06971=1062.160,3.732,432.100,171.833,27.398,155.079
C06972=1062.154,3.482,432.114,171.831,27.395,155.079
C06973=1062.148,3.233,432.128,171.829,27.393,155.079
C06974=1062.142,2.983,432.143,171.828,27.390,155.078
C06975=1062.135,2.734,432.158,171.827,27.388,155.078
C06976=1062.130,2.484,432.172,171.826,27.385,155.078
C06977=1062.124,2.234,432.187,171.824,27.383,155.077
C06978=1062.118,1.985,432.202,171.823,27.380,155.077
C06979=1062.111,1.736,432.217,171.821,27.378,155.077
C06980=1062.106,1.486,432.231,171.819,27.376,155.076
C06981=1062.100,1.236,432.245,171.818,27.373,155.076
C06982=1062.094,0.988,432.260,171.816,27.371,155.076
C06983=1062.087,0.738,432.275,171.815,27.368,155.076
C06984=1062.082,0.488,432.289,171.813,27.366,155.075
C06985=1062.076,0.239,432.304,171.812,27.363,155.075
C06986=1062.070,-0.010,432.318,171.810,27.361,155.075
C06987=1062.064,-0.261,432.333,171.810,27.358,155.074
C06988=1062.058,-0.510,432.347,171.808,27.356,155.074
C06989=1062.052,-0.759,432.362,171.806,27.354,155.074
C06990=1062.046,-1.009,432.376,171.805,27.351,155.073
C06991=1062.040,-1.258,432.391,171.803,27.349,155.073
C06992=1062.034,-1.507,432.406,171.802,27.346,155.073
C06993=1062.027,-1.788,432.421,171.800,27.344,155.072
C06994=1062.021,-2.070,432.438,171.799,27.341,155.072
C06995=1062.014,-2.350,432.454,171.797,27.338,155.072
C06996=1062.007,-2.631,432.470,171.795,27.335,155.071
C06997=1062.000,-2.881,432.485,171.793,27.333,155.071
C06998=1061.995,-3.131,432.499,171.793,27.331,155.071
C06999=1061.988,-3.380,432.514,171.791,27.328,155.070
C07000=1061.983,-3.630,432.527,171.789,27.326,155.070
C07001=1061.977,-3.880,432.542,171.788,27.323,155.070
C07002=1061.970,-4.128,432.556,171.786,27.321,155.069
C07003=1061.964,-4.379,432.571,171.785,27.319,155.069
C07004=1061.958,-4.627,432.585,171.783,27.316,155.069
C07005=1061.951,-4.877,432.599,171.782,27.314,155.069
C07006=1061.946,-5.126,432.613,171.780,27.312,155.068
C07007=1061.939,-5.377,432.628,171.778,27.309,155.068
C07008=1061.934,-5.626,432.642,171.777,27.307,155.068
C07009=1061.927,-5.876,432.656,171.775,27.304,155.067
C07010=1061.921,-6.125,432.670,171.774,27.302,155.067
C07011=1061.915,-6.375,432.685,171.772,27.300,155.067
C07012=1061.909,-6.624,432.698,171.771,27.298,155.067
C07013=1061.902,-6.874,432.713,171.770,27.296,155.066
C07014=1061.897,-7.123,432.727,171.768,27.293,155.066
C07015=1061.890,-7.373,432.741,171.767,27.290,155.066
C07016=1061.884,-7.622,432.755,171.765,27.288,155.065
C07017=1061.879,-7.871,432.770,171.764,27.286,155.065
C07018=1061.872,-8.121,432.783,171.762,27.284,155.065
C07019=1061.866,-8.371,432.797,171.760,27.281,155.065
C07020=1061.860,-8.620,432.812,171.759,27.279,155.064
C07021=1061.854,-8.870,432.825,171.757,27.277,155.064
C07022=1061.847,-9.119,432.840,171.756,27.274,155.064
C07023=1061.842,-9.369,432.854,171.754,27.272,155.063
C07024=1061.836,-9.618,432.867,171.753,27.269,155.063
C07025=1061.829,-9.868,432.882,171.751,27.267,155.063
C07026=1061.824,-10.117,432.896,171.749,27.265,155.063
C07027=1061.817,-10.367,432.910,171.749,27.263,155.062
C07028=1061.811,-10.616,432.924,171.747,27.261,155.062
C07029=1061.806,-10.866,432.938,171.746,27.258,155.062
C07030=1061.799,-11.116,432.952,171.744,27.256,155.062
C07031=1061.793,-11.365,432.966,171.743,27.253,155.061
C07032=1061.787,-11.615,432.981,171.741,27.251,155.061
C07033=1061.781,-11.864,432.994,171.739,27.249,155.061
C07034=1061.775,-12.113,433.009,171.738,27.246,155.060
C07035=1061.768,-12.363,433.022,171.736,27.244,155.060
C07036=1061.763,-12.613,433.036,171.735,27.242,155.060
C07037=1061.757,-12.862,433.050,171.733,27.239,155.060
C07038=1061.750,-13.112,433.064,171.732,27.237,155.059
C07039=1061.745,-13.361,433.078,171.730,27.235,155.059
C07040=1061.739,-13.611,433.092,171.728,27.232,155.059
C07041=1061.732,-13.861,433.106,171.727,27.230,155.058
C07042=1061.727,-14.110,433.120,171.725,27.227,155.058
C07043=1061.720,-14.359,433.133,171.724,27.225,155.058
C07044=1061.714,-14.609,433.148,171.723,27.223,155.058
C07045=1061.709,-14.859,433.162,171.722,27.221,155.057
C07046=1061.703,-15.108,433.175,171.720,27.219,155.057
C07047=1061.696,-15.358,433.190,171.718,27.216,155.057
C07048=1061.690,-15.607,433.203,171.717,27.214,155.056
C07049=1061.684,-15.856,433.216,171.715,27.212,155.056
C07050=1061.678,-16.107,433.231,171.714,27.209,155.056
C07051=1061.671,-16.356,433.244,171.712,27.207,155.056
C07052=1061.665,-16.606,433.258,171.710,27.205,155.055
C07053=1061.659,-16.855,433.272,171.709,27.203,155.055
C07054=1061.653,-17.104,433.286,171.707,27.200,155.055
C07055=1061.647,-17.354,433.300,171.706,27.198,155.055
C07056=1061.640,-17.604,433.313,171.704,27.196,155.054
C07057=1061.634,-17.883,433.328,171.703,27.194,155.054
C07058=1061.627,-18.163,433.343,171.701,27.191,155.054
C07059=1061.620,-18.442,433.359,171.700,27.188,155.053
C07060=1061.613,-18.721,433.374,171.697,27.186,155.053
C07061=1061.608,-18.971,433.388,171.695,27.184,155.053
C07062=1061.601,-19.221,433.401,171.694,27.181,155.053
C07063=1061.595,-19.470,433.415,171.692,27.179,155.052
C07064=1061.589,-19.719,433.429,171.692,27.177,155.052
C07065=1061.582,-19.969,433.442,171.690,27.175,155.052
C07066=1061.577,-20.219,433.456,171.688,27.173,155.052
C07067=1061.571,-20.468,433.469,171.687,27.171,155.051
C07068=1061.564,-20.717,433.483,171.685,27.168,155.051
C07069=1061.558,-20.968,433.497,171.684,27.166,155.051
C07070=1061.552,-21.217,433.510,171.682,27.164,155.051
C07071=1061.546,-21.466,433.523,171.680,27.162,155.050
C07072=1061.540,-21.716,433.537,171.679,27.159,155.050
C07073=1061.534,-21.966,433.551,171.677,27.157,155.050
C07074=1061.527,-22.215,433.564,171.676,27.155,155.050
C07075=1061.522,-22.465,433.578,171.674,27.152,155.049
C07076=1061.516,-22.714,433.591,171.673,27.150,155.049
C07077=1061.509,-22.964,433.605,171.671,27.148,155.049
C07078=1061.503,-23.213,433.619,171.669,27.146,155.049
C07079=1061.497,-23.463,433.632,171.668,27.144,155.048
C07080=1061.491,-23.712,433.645,171.666,27.142,155.048
C07081=1061.486,-23.962,433.659,171.665,27.139,155.048
C07082=1061.479,-24.212,433.673,171.663,27.137,155.047
C07083=1061.472,-24.461,433.686,171.661,27.135,155.047
C07084=1061.467,-24.711,433.699,171.660,27.132,155.047
C07085=1061.461,-24.960,433.712,171.658,27.130,155.047
C07086=1061.455,-25.210,433.726,171.657,27.128,155.046
C07087=1061.449,-25.460,433.740,171.655,27.126,155.046
C07088=1061.443,-25.709,433.753,171.653,27.124,155.046
C07089=1061.436,-25.958,433.767,171.652,27.122,155.046
C07090=1061.431,-26.208,433.780,171.650,27.119,155.045
C07091=1061.425,-26.458,433.793,171.649,27.117,155.045
C07092=1061.419,-26.707,433.806,171.648,27.115,155.045
C07093=1061.413,-26.957,433.820,171.647,27.113,155.045
C07094=1061.406,-27.207,433.834,171.645,27.111,155.045
C07095=1061.400,-27.456,433.847,171.643,27.109,155.044
C07096=1061.394,-27.705,433.860,171.642,27.106,155.044
C07097=1061.388,-27.955,433.873,171.640,27.104,155.044
C07098=1061.381,-28.205,433.886,171.639,27.102,155.044
C07099=1061.375,-28.454,433.900,171.637,27.100,155.043
C07100=1061.369,-28.703,433.913,171.635,27.098,155.043
C07101=1061.363,-28.953,433.926,171.634,27.096,155.043
C07102=1061.357,-29.203,433.939,171.632,27.094,155.043
C07103=1061.351,-29.452,433.953,171.631,27.092,155.042
C07104=1061.345,-29.702,433.966,171.629,27.089,155.042
C07105=1061.339,-29.952,433.979,171.627,27.088,155.042
C07106=1061.332,-30.201,433.992,171.626,27.085,155.042
C07107=1061.326,-30.451,434.005,171.624,27.083,155.041
C07108=1061.320,-30.700,434.018,171.623,27.081,155.041
C07109=1061.314,-30.950,434.031,171.621,27.079,155.041
C07110=1061.308,-31.199,434.044,171.619,27.077,155.041
C07111=1061.301,-31.450,434.057,171.618,27.074,155.040
C07112=1061.295,-31.699,434.071,171.616,27.073,155.040
C07113=1061.289,-31.948,434.084,171.615,27.070,155.040
C07114=1061.283,-32.198,434.096,171.613,27.068,155.040
C07115=1061.278,-32.448,434.110,171.611,27.066,155.040
C07116=1061.271,-32.697,434.124,171.610,27.064,155.039
C07117=1061.265,-32.947,434.136,171.608,27.062,155.039
C07118=1061.259,-33.196,434.149,171.607,27.060,155.039
C07119=1061.253,-33.446,434.162,171.605,27.058,155.039
C07120=1061.247,-33.695,434.175,171.603,27.056,155.038
C07121=1061.240,-33.974,434.190,171.602,27.053,155.038
C07122=1061.233,-34.253,434.204,171.600,27.051,155.038
C07123=1061.226,-34.532,434.219,171.598,27.048,155.038
C07124=1061.219,-34.809,434.233,171.596,27.046,155.037
C07125=1061.213,-35.059,434.246,171.595,27.044,155.037
C07126=1061.207,-35.309,434.259,171.593,27.042,155.037
C07127=1061.201,-35.558,434.272,171.591,27.040,155.037
C07128=1061.195,-35.808,434.285,171.590,27.038,155.037
C07129=1061.189,-36.057,434.298,171.588,27.036,155.036
C07130=1061.183,-36.307,434.311,171.586,27.034,155.036
C07131=1061.177,-36.556,434.324,171.585,27.032,155.036
C07132=1061.170,-36.807,434.337,171.583,27.030,155.036
C07133=1061.164,-37.056,434.350,171.582,27.027,155.035
C07134=1061.158,-37.306,434.363,171.580,27.026,155.035
C07135=1061.152,-37.555,434.376,171.578,27.023,155.035
C07136=1061.146,-37.805,434.389,171.577,27.021,155.035
C07137=1061.140,-38.055,434.401,171.575,27.019,155.035
C07138=1061.134,-38.304,434.415,171.574,27.017,155.034
C07139=1061.128,-38.554,434.427,171.572,27.015,155.034
C07140=1061.122,-38.803,434.440,171.570,27.013,155.034
C07141=1061.116,-39.053,434.453,171.569,27.011,155.034
C07142=1061.110,-39.302,434.466,171.567,27.009,155.033
C07143=1061.104,-39.552,434.479,171.566,27.007,155.033
C07144=1061.098,-39.802,434.491,171.564,27.005,155.033
C07145=1061.091,-40.051,434.504,171.562,27.003,155.033
C07146=1061.085,-40.301,434.517,171.561,27.001,155.033
C07147=1061.079,-40.550,434.530,171.559,26.999,155.033
C07148=1061.073,-40.800,434.542,171.557,26.997,155.032
C07149=1061.067,-41.050,434.555,171.556,26.995,155.032
C07150=1061.060,-41.299,434.568,171.554,26.993,155.032
C07151=1061.054,-41.549,434.580,171.553,26.991,155.032
C07152=1061.048,-41.799,434.593,171.551,26.989,155.031
C07153=1061.042,-42.048,434.606,171.549,26.987,155.031
C07154=1061.035,-42.298,434.618,171.548,26.985,155.031
C07155=1061.029,-42.547,434.631,171.546,26.983,155.031
C07156=1061.023,-42.797,434.644,171.545,26.981,155.031
C07157=1061.017,-43.047,434.656,171.543,26.979,155.030
C07158=1061.011,-43.297,434.669,171.541,26.977,155.030
C07159=1061.005,-43.546,434.681,171.540,26.975,155.030
C07160=1060.999,-43.795,434.694,171.538,26.973,155.030
C07161=1060.993,-44.045,434.707,171.536,26.971,155.030
C07162=1060.987,-44.294,434.719,171.535,26.969,155.030
C07163=1060.980,-44.543,434.732,171.533,26.967,155.029
C07164=1060.974,-44.793,434.744,171.531,26.965,155.029
C07165=1060.969,-45.043,434.757,171.530,26.963,155.029
C07166=1060.963,-45.293,434.769,171.528,26.961,155.029
C07167=1060.956,-45.543,434.781,171.527,26.960,155.029
C07168=1060.950,-45.792,434.794,171.525,26.957,155.028
C07169=1060.944,-46.042,434.807,171.523,26.956,155.028
C07170=1060.938,-46.292,434.820,171.522,26.953,155.028
C07171=1060.931,-46.541,434.832,171.520,26.952,155.028
C07172=1060.925,-46.791,434.844,171.518,26.950,155.028
C07173=1060.919,-47.040,434.857,171.517,26.948,155.027
C07174=1060.914,-47.289,434.870,171.515,26.946,155.027
C07175=1060.907,-47.539,434.881,171.514,26.944,155.027
C07176=1060.901,-47.789,434.894,171.512,26.942,155.027
C07177=1060.895,-48.039,434.907,171.510,26.940,155.027
C07178=1060.890,-48.289,434.919,171.509,26.938,155.026
C07179=1060.883,-48.538,434.932,171.507,26.936,155.026
C07180=1060.877,-48.788,434.944,171.505,26.934,155.026
C07181=1060.871,-49.037,434.957,171.504,26.932,155.026
C07182=1060.865,-49.286,434.969,171.502,26.930,155.026
C07183=1060.859,-49.536,434.981,171.501,26.928,155.025
C07184=1060.853,-49.786,434.994,171.499,26.926,155.025
C07185=1060.846,-50.065,435.007,171.496,26.924,155.025
C07186=1060.839,-50.343,435.021,171.495,26.922,155.025
C07187=1060.833,-50.623,435.035,171.493,26.920,155.025
C07188=1060.825,-50.902,435.049,171.492,26.918,155.024
C07189=1060.819,-51.151,435.061,171.490,26.916,155.024
C07190=1060.812,-51.401,435.073,171.488,26.915,155.024
C07191=1060.806,-51.651,435.086,171.487,26.913,155.024
C07192=1060.800,-51.901,435.098,171.485,26.911,155.024
C07193=1060.794,-52.150,435.110,171.483,26.909,155.024
C07194=1060.788,-52.399,435.122,171.481,26.907,155.024
C07195=1060.781,-52.649,435.134,171.479,26.905,155.023
C07196=1060.775,-52.899,435.146,171.477,26.904,155.023
C07197=1060.768,-53.148,435.158,171.476,26.902,155.023
C07198=1060.762,-53.398,435.171,171.474,26.900,155.023
C07199=1060.756,-53.648,435.183,171.473,26.898,155.023
C07200=1060.750,-53.897,435.194,171.471,26.896,155.023
C07201=1060.744,-54.147,435.206,171.469,26.894,155.022
C07202=1060.738,-54.397,435.218,171.468,26.893,155.022
C07203=1060.732,-54.647,435.231,171.466,26.891,155.022
C07204=1060.725,-54.896,435.243,171.464,26.889,155.022
C07205=1060.718,-55.146,435.255,171.463,26.887,155.022
C07206=1060.712,-55.396,435.267,171.461,26.886,155.022
C07207=1060.706,-55.644,435.279,171.459,26.884,155.022
C07208=1060.700,-55.894,435.291,171.458,26.882,155.021
C07209=1060.694,-56.144,435.303,171.456,26.880,155.021
C07210=1060.687,-56.393,435.315,171.454,26.878,155.021
C07211=1060.682,-56.644,435.327,171.453,26.877,155.021
C07212=1060.676,-56.893,435.339,171.451,26.875,155.021
C07213=1060.669,-57.142,435.351,171.449,26.873,155.021
C07214=1060.663,-57.392,435.363,171.448,26.871,155.020
C07215=1060.656,-57.642,435.375,171.446,26.870,155.020
C07216=1060.650,-57.891,435.387,171.444,26.868,155.020
C07217=1060.645,-58.141,435.399,171.443,26.866,155.020
C07218=1060.638,-58.391,435.410,171.441,26.865,155.020
C07219=1060.632,-58.641,435.423,171.439,26.863,155.020
C07220=1060.625,-58.890,435.435,171.438,26.861,155.020
C07221=1060.619,-59.139,435.447,171.436,26.859,155.019
C07222=1060.614,-59.390,435.458,171.433,26.857,155.019
C07223=1060.607,-59.639,435.470,171.432,26.856,155.019
C07224=1060.601,-59.889,435.482,171.430,26.854,155.019
C07225=1060.595,-60.138,435.495,171.428,26.852,155.019
C07226=1060.589,-60.388,435.506,171.427,26.851,155.019
C07227=1060.582,-60.638,435.518,171.425,26.849,155.019
C07228=1060.577,-60.887,435.530,171.423,26.847,155.018
C07229=1060.570,-61.137,435.542,171.422,26.845,155.018
C07230=1060.564,-61.387,435.553,171.420,26.844,155.018
C07231=1060.558,-61.637,435.566,171.418,26.842,155.018
C07232=1060.552,-61.885,435.577,171.417,26.840,155.018
C07233=1060.545,-62.135,435.589,171.415,26.838,155.018
C07234=1060.539,-62.385,435.600,171.413,26.837,155.018
C07235=1060.534,-62.634,435.613,171.412,26.835,155.017
C07236=1060.527,-62.884,435.625,171.410,26.833,155.017
C07237=1060.521,-63.134,435.636,171.408,26.832,155.017
C07238=1060.515,-63.383,435.648,171.407,26.830,155.017
C07239=1060.509,-63.633,435.660,171.405,26.828,155.017
C07240=1060.502,-63.883,435.671,171.403,26.826,155.017
C07241=1060.497,-64.132,435.683,171.402,26.825,155.017
C07242=1060.491,-64.382,435.695,171.400,26.823,155.016
C07243=1060.484,-64.632,435.707,171.399,26.821,155.016
C07244=1060.478,-64.881,435.718,171.397,26.820,155.016
C07245=1060.472,-65.131,435.730,171.395,26.818,155.016
C07246=1060.466,-65.380,435.742,171.393,26.816,155.016
C07247=1060.460,-65.630,435.753,171.391,26.814,155.016
C07248=1060.454,-65.880,435.765,171.389,26.812,155.016
C07249=1060.447,-66.160,435.779,171.388,26.811,155.016
C07250=1060.441,-66.440,435.791,171.386,26.809,155.015
C07251=1060.433,-66.721,435.804,171.383,26.807,155.015
C07252=1060.427,-67.001,435.817,171.382,26.805,155.015
C07253=1060.421,-67.251,435.829,171.380,26.803,155.015
C07254=1060.415,-67.500,435.840,171.378,26.802,155.015
C07255=1060.408,-67.750,435.852,171.377,26.800,155.015
C07256=1060.402,-68.000,435.863,171.375,26.798,155.015
C07257=1060.397,-68.249,435.876,171.373,26.797,155.014
C07258=1060.390,-68.499,435.888,171.372,26.795,155.014
C07259=1060.384,-68.748,435.898,171.370,26.794,155.014
C07260=1060.378,-68.999,435.910,171.368,26.792,155.014
C07261=1060.373,-69.248,435.922,171.367,26.790,155.014
C07262=1060.366,-69.498,435.933,171.365,26.789,155.014
C07263=1060.360,-69.747,435.945,171.363,26.787,155.014
C07264=1060.354,-69.997,435.956,171.362,26.785,155.014
C07265=1060.348,-70.247,435.969,171.360,26.783,155.013
C07266=1060.342,-70.496,435.979,171.358,26.782,155.013
C07267=1060.336,-70.746,435.991,171.356,26.780,155.013
C07268=1060.330,-70.996,436.002,171.354,26.778,155.013
C07269=1060.324,-71.246,436.013,171.352,26.777,155.013
C07270=1060.318,-71.495,436.026,171.351,26.775,155.013
C07271=1060.312,-71.745,436.037,171.349,26.773,155.013
C07272=1060.306,-71.994,436.049,171.347,26.772,155.013
C07273=1060.300,-72.244,436.060,171.346,26.770,155.013
C07274=1060.295,-72.494,436.071,171.344,26.769,155.012
C07275=1060.288,-72.744,436.083,171.342,26.767,155.012
C07276=1060.282,-72.993,436.094,171.341,26.765,155.012
C07277=1060.275,-73.243,436.106,171.339,26.764,155.012
C07278=1060.270,-73.492,436.117,171.337,26.762,155.012
C07279=1060.264,-73.743,436.129,171.335,26.761,155.012
C07280=1060.258,-73.992,436.140,171.334,26.759,155.012
C07281=1060.252,-74.242,436.152,171.332,26.758,155.012
C07282=1060.246,-74.491,436.162,171.330,26.756,155.012
C07283=1060.240,-74.741,436.174,171.329,26.754,155.011
